   1:  PR[91] = PR[90];
   1:  PR[91,1] = PR[90,1] + 58.395;
   1:  PR[91,2] = PR[90,2] + 13.062;
   1:  PR[91,3] = PR[90,3] + 26.195;
   1:  PR[92] = PR[91];
   1:  PR[92,3] = PR[92,3] + 20;
   1:J PR[92] 10% FINE;
   1:L PR[91] R[100]mm/sec CNT100;
   1:  CALL LASER_DRAHT_START;
   1:  PR[91,1] = PR[90,1] + 56.578;
   1:  PR[91,2] = PR[90,2] + 11.493;
   1:L PR[91] R[100]mm/sec CNT100;
   1:  PR[91,1] = PR[90,1] + 55.757;
   1:  PR[91,2] = PR[90,2] + 10.310;
   1:L PR[91] R[100]mm/sec CNT100;
   1:  PR[91,1] = PR[90,1] + 53.974;
   1:  PR[91,2] = PR[90,2] + 7.827;
   1:L PR[91] R[100]mm/sec CNT100;
   1:  PR[91,1] = PR[90,1] + 52.340;
   1:  PR[91,2] = PR[90,2] + 3.681;
   1:L PR[91] R[100]mm/sec CNT100;
   1:  PR[91,1] = PR[90,1] + 52.290;
   1:  PR[91,2] = PR[90,2] + 3.287;
   1:L PR[91] R[100]mm/sec CNT100;
   1:  PR[91,1] = PR[90,1] + 52.250;
   1:  PR[91,2] = PR[90,2] + 2.641;
   1:L PR[91] R[100]mm/sec CNT100;
   1:  PR[91,1] = PR[90,1] + 51.813;
   1:  PR[91,2] = PR[90,2] + -0.787;
   1:L PR[91] R[100]mm/sec CNT100;
   1:  PR[91,1] = PR[90,1] + 51.829;
   1:  PR[91,2] = PR[90,2] + -1.013;
   1:L PR[91] R[100]mm/sec CNT100;
   1:  PR[91,1] = PR[90,1] + 52.341;
   1:  PR[91,2] = PR[90,2] + -5.143;
   1:L PR[91] R[100]mm/sec CNT100;
   1:  PR[91,1] = PR[90,1] + 53.979;
   1:  PR[91,2] = PR[90,2] + -9.300;
   1:L PR[91] R[100]mm/sec CNT100;
   1:  PR[91,1] = PR[90,1] + 54.599;
   1:  PR[91,2] = PR[90,2] + -10.189;
   1:L PR[91] R[100]mm/sec CNT100;
   1:  PR[91,1] = PR[90,1] + 56.578;
   1:  PR[91,2] = PR[90,2] + -12.957;
   1:L PR[91] R[100]mm/sec CNT100;
   1:  PR[91,1] = PR[90,1] + 57.989;
   1:  PR[91,2] = PR[90,2] + -14.220;
   1:L PR[91] R[100]mm/sec CNT100;
   1:  PR[91,1] = PR[90,1] + 59.963;
   1:  PR[91,2] = PR[90,2] + -15.936;
   1:L PR[91] R[100]mm/sec CNT100;
   1:  PR[91,1] = PR[90,1] + 62.463;
   1:  PR[91,2] = PR[90,2] + -17.317;
   1:L PR[91] R[100]mm/sec CNT100;
   1:  PR[91,1] = PR[90,1] + 63.933;
   1:  PR[91,2] = PR[90,2] + -18.100;
   1:L PR[91] R[100]mm/sec CNT100;
   1:  PR[91,1] = PR[90,1] + 67.611;
   1:  PR[91,2] = PR[90,2] + -19.179;
   1:L PR[91] R[100]mm/sec CNT100;
   1:  PR[91,1] = PR[90,1] + 68.271;
   1:  PR[91,2] = PR[90,2] + -19.362;
   1:L PR[91] R[100]mm/sec CNT100;
   1:  PR[91,1] = PR[90,1] + 72.776;
   1:  PR[91,2] = PR[90,2] + -19.685;
   1:L PR[91] R[100]mm/sec CNT100;
   1:  PR[91,1] = PR[90,1] + 77.061;
   1:  PR[91,2] = PR[90,2] + -19.105;
   1:L PR[91] R[100]mm/sec CNT100;
   1:  PR[91,1] = PR[90,1] + 81.078;
   1:  PR[91,2] = PR[90,2] + -17.631;
   1:L PR[91] R[100]mm/sec CNT100;
   1:  PR[91,1] = PR[90,1] + 84.652;
   1:  PR[91,2] = PR[90,2] + -15.336;
   1:L PR[91] R[100]mm/sec CNT100;
   1:  PR[91,1] = PR[90,1] + 87.617;
   1:  PR[91,2] = PR[90,2] + -12.341;
   1:L PR[91] R[100]mm/sec CNT100;
   1:  PR[91,1] = PR[90,1] + 89.839;
   1:  PR[91,2] = PR[90,2] + -8.790;
   1:L PR[91] R[100]mm/sec CNT100;
   1:  PR[91,1] = PR[90,1] + 90.385;
   1:  PR[91,2] = PR[90,2] + -7.237;
   1:L PR[91] R[100]mm/sec CNT100;
   1:  PR[91,1] = PR[90,1] + 91.211;
   1:  PR[91,2] = PR[90,2] + -4.857;
   1:L PR[91] R[100]mm/sec CNT100;
   1:  PR[91,1] = PR[90,1] + 91.419;
   1:  PR[91,2] = PR[90,2] + -3.053;
   1:L PR[91] R[100]mm/sec CNT100;
   1:  PR[91,1] = PR[90,1] + 91.779;
   1:  PR[91,2] = PR[90,2] + -0.692;
   1:L PR[91] R[100]mm/sec CNT100;
   1:  PR[91,1] = PR[90,1] + 91.764;
   1:  PR[91,2] = PR[90,2] + -0.562;
   1:L PR[91] R[100]mm/sec CNT100;
   1:  PR[91,1] = PR[90,1] + 91.478;
   1:  PR[91,2] = PR[90,2] + 0.980;
   1:L PR[91] R[100]mm/sec CNT100;
   1:  PR[91,1] = PR[90,1] + 91.210;
   1:  PR[91,2] = PR[90,2] + 3.401;
   1:L PR[91] R[100]mm/sec CNT100;
   1:  PR[91,1] = PR[90,1] + 89.838;
   1:  PR[91,2] = PR[90,2] + 7.333;
   1:L PR[91] R[100]mm/sec CNT100;
   1:  PR[91,1] = PR[90,1] + 87.617;
   1:  PR[91,2] = PR[90,2] + 10.882;
   1:L PR[91] R[100]mm/sec CNT100;
   1:  PR[91,1] = PR[90,1] + 84.658;
   1:  PR[91,2] = PR[90,2] + 13.872;
   1:L PR[91] R[100]mm/sec CNT100;
   1:  PR[91,1] = PR[90,1] + 83.729;
   1:  PR[91,2] = PR[90,2] + 14.458;
   1:L PR[91] R[100]mm/sec CNT100;
   1:  PR[91,1] = PR[90,1] + 81.076;
   1:  PR[91,2] = PR[90,2] + 16.173;
   1:L PR[91] R[100]mm/sec CNT100;
   1:  PR[91,1] = PR[90,1] + 77.061;
   1:  PR[91,2] = PR[90,2] + 17.647;
   1:L PR[91] R[100]mm/sec CNT100;
   1:  PR[91,1] = PR[90,1] + 72.779;
   1:  PR[91,2] = PR[90,2] + 18.226;
   1:L PR[91] R[100]mm/sec CNT100;
   1:  PR[91,1] = PR[90,1] + 68.646;
   1:  PR[91,2] = PR[90,2] + 17.919;
   1:L PR[91] R[100]mm/sec CNT100;
   1:  PR[91,1] = PR[90,1] + 68.271;
   1:  PR[91,2] = PR[90,2] + 17.899;
   1:L PR[91] R[100]mm/sec CNT100;
   1:  PR[91,1] = PR[90,1] + 64.923;
   1:  PR[91,2] = PR[90,2] + 16.906;
   1:L PR[91] R[100]mm/sec CNT100;
   1:  PR[91,1] = PR[90,1] + 63.934;
   1:  PR[91,2] = PR[90,2] + 16.636;
   1:L PR[91] R[100]mm/sec CNT100;
   1:  PR[91,1] = PR[90,1] + 61.478;
   1:  PR[91,2] = PR[90,2] + 15.271;
   1:L PR[91] R[100]mm/sec CNT100;
   1:  PR[91,1] = PR[90,1] + 59.964;
   1:  PR[91,2] = PR[90,2] + 14.472;
   1:L PR[91] R[100]mm/sec CNT100;
   1:  PR[91,1] = PR[90,1] + 58.395;
   1:  PR[91,2] = PR[90,2] + 13.062;
   1:L PR[91] R[100]mm/sec CNT100TB   .50sec,CALL END_PUD;
   1:  PR[92] = PR[91];
   1:  PR[92,3] = PR[92,3] + 20;
   1:J PR[92] 10% FINE;
   1:  PR[91,1] = PR[90,1] + 41.160;
   1:  PR[91,2] = PR[90,2] + 8.184;
   1:  PR[92] = PR[91];
   1:  PR[92,3] = PR[92,3] + 20;
   1:J PR[92] 10% FINE;
   1:L PR[91] R[100]mm/sec CNT100;
   1:  CALL LASER_DRAHT_START;
   1:  PR[91,1] = PR[90,1] + 40.947;
   1:  PR[91,2] = PR[90,2] + 8.666;
   1:L PR[91] R[100]mm/sec CNT100;
   1:  PR[91,1] = PR[90,1] + 38.341;
   1:  PR[91,2] = PR[90,2] + 12.079;
   1:L PR[91] R[100]mm/sec CNT100;
   1:  PR[91,1] = PR[90,1] + 37.898;
   1:  PR[91,2] = PR[90,2] + 12.643;
   1:L PR[91] R[100]mm/sec CNT100;
   1:  PR[91,1] = PR[90,1] + 33.979;
   1:  PR[91,2] = PR[90,2] + 15.652;
   1:L PR[91] R[100]mm/sec CNT100;
   1:  PR[91,1] = PR[90,1] + 30.208;
   1:  PR[91,2] = PR[90,2] + 17.229;
   1:L PR[91] R[100]mm/sec CNT100;
   1:  PR[91,1] = PR[90,1] + 29.432;
   1:  PR[91,2] = PR[90,2] + 17.545;
   1:L PR[91] R[100]mm/sec CNT100;
   1:  PR[91,1] = PR[90,1] + 24.528;
   1:  PR[91,2] = PR[90,2] + 18.204;
   1:L PR[91] R[100]mm/sec CNT100;
   1:  PR[91,1] = PR[90,1] + 19.621;
   1:  PR[91,2] = PR[90,2] + 17.571;
   1:L PR[91] R[100]mm/sec CNT100;
   1:  PR[91,1] = PR[90,1] + 16.027;
   1:  PR[91,2] = PR[90,2] + 16.100;
   1:L PR[91] R[100]mm/sec CNT100;
   1:  PR[91,1] = PR[90,1] + 15.045;
   1:  PR[91,2] = PR[90,2] + 15.693;
   1:L PR[91] R[100]mm/sec CNT100;
   1:  PR[91,1] = PR[90,1] + 11.102;
   1:  PR[91,2] = PR[90,2] + 12.688;
   1:L PR[91] R[100]mm/sec CNT100;
   1:  PR[91,1] = PR[90,1] + 8.076;
   1:  PR[91,2] = PR[90,2] + 8.763;
   1:L PR[91] R[100]mm/sec CNT100;
   1:  PR[91,1] = PR[90,1] + 6.171;
   1:  PR[91,2] = PR[90,2] + 4.186;
   1:L PR[91] R[100]mm/sec CNT100;
   1:  PR[91,1] = PR[90,1] + 5.520;
   1:  PR[91,2] = PR[90,2] + -0.729;
   1:L PR[91] R[100]mm/sec CNT100;
   1:  PR[91,1] = PR[90,1] + 6.171;
   1:  PR[91,2] = PR[90,2] + -5.646;
   1:L PR[91] R[100]mm/sec CNT100;
   1:  PR[91,1] = PR[90,1] + 8.077;
   1:  PR[91,2] = PR[90,2] + -10.225;
   1:L PR[91] R[100]mm/sec CNT100;
   1:  PR[91,1] = PR[90,1] + 11.105;
   1:  PR[91,2] = PR[90,2] + -14.150;
   1:L PR[91] R[100]mm/sec CNT100;
   1:  PR[91,1] = PR[90,1] + 15.047;
   1:  PR[91,2] = PR[90,2] + -17.153;
   1:L PR[91] R[100]mm/sec CNT100;
   1:  PR[91,1] = PR[90,1] + 19.631;
   1:  PR[91,2] = PR[90,2] + -19.033;
   1:L PR[91] R[100]mm/sec CNT100;
   1:  PR[91,1] = PR[90,1] + 20.613;
   1:  PR[91,2] = PR[90,2] + -19.162;
   1:L PR[91] R[100]mm/sec CNT100;
   1:  PR[91,1] = PR[90,1] + 24.534;
   1:  PR[91,2] = PR[90,2] + -19.663;
   1:L PR[91] R[100]mm/sec CNT100;
   1:  PR[91,1] = PR[90,1] + 29.431;
   1:  PR[91,2] = PR[90,2] + -19.003;
   1:L PR[91] R[100]mm/sec CNT100;
   1:  PR[91,1] = PR[90,1] + 33.994;
   1:  PR[91,2] = PR[90,2] + -17.103;
   1:L PR[91] R[100]mm/sec CNT100;
   1:  PR[91,1] = PR[90,1] + 34.610;
   1:  PR[91,2] = PR[90,2] + -16.637;
   1:L PR[91] R[100]mm/sec CNT100;
   1:  PR[91,1] = PR[90,1] + 37.894;
   1:  PR[91,2] = PR[90,2] + -14.104;
   1:L PR[91] R[100]mm/sec CNT100;
   1:  PR[91,1] = PR[90,1] + 40.936;
   1:  PR[91,2] = PR[90,2] + -10.139;
   1:L PR[91] R[100]mm/sec CNT100;
   1:  PR[91,1] = PR[90,1] + 42.580;
   1:  PR[91,2] = PR[90,2] + -6.157;
   1:L PR[91] R[100]mm/sec CNT100;
   1:  PR[91,1] = PR[90,1] + 42.727;
   1:  PR[91,2] = PR[90,2] + -5.828;
   1:L PR[91] R[100]mm/sec CNT100;
   1:  PR[91,1] = PR[90,1] + 42.869;
   1:  PR[91,2] = PR[90,2] + -5.270;
   1:L PR[91] R[100]mm/sec CNT100;
   1:  PR[91,1] = PR[90,1] + 43.360;
   1:  PR[91,2] = PR[90,2] + -1.542;
   1:L PR[91] R[100]mm/sec CNT100;
   1:  PR[91,1] = PR[90,1] + 43.428;
   1:  PR[91,2] = PR[90,2] + -0.772;
   1:L PR[91] R[100]mm/sec CNT100;
   1:  PR[91,1] = PR[90,1] + 42.958;
   1:  PR[91,2] = PR[90,2] + 2.798;
   1:L PR[91] R[100]mm/sec CNT100;
   1:  PR[91,1] = PR[90,1] + 42.866;
   1:  PR[91,2] = PR[90,2] + 3.815;
   1:L PR[91] R[100]mm/sec CNT100;
   1:  PR[91,1] = PR[90,1] + 42.702;
   1:  PR[91,2] = PR[90,2] + 4.446;
   1:L PR[91] R[100]mm/sec CNT100;
   1:  PR[91,1] = PR[90,1] + 41.160;
   1:  PR[91,2] = PR[90,2] + 8.184;
   1:L PR[91] R[100]mm/sec CNT100TB   .50sec,CALL END_PUD;
   1:  PR[92] = PR[91];
   1:  PR[92,3] = PR[92,3] + 20;
   1:J PR[92] 10% FINE;
   1:  PR[91,1] = PR[90,1] + -27.836;
   1:  PR[91,2] = PR[90,2] + -18.849;
   1:  PR[92] = PR[91];
   1:  PR[92,3] = PR[92,3] + 20;
   1:J PR[92] 10% FINE;
   1:L PR[91] R[100]mm/sec CNT100;
   1:  CALL LASER_DRAHT_START;
   1:  PR[91,1] = PR[90,1] + -25.440;
   1:  PR[91,2] = PR[90,2] + -19.136;
   1:L PR[91] R[100]mm/sec CNT100;
   1:  PR[91,1] = PR[90,1] + -23.651;
   1:  PR[91,2] = PR[90,2] + -19.368;
   1:L PR[91] R[100]mm/sec CNT100;
   1:  PR[91,1] = PR[90,1] + -21.486;
   1:  PR[91,2] = PR[90,2] + -19.143;
   1:L PR[91] R[100]mm/sec CNT100;
   1:  PR[91,1] = PR[90,1] + -19.442;
   1:  PR[91,2] = PR[90,2] + -18.953;
   1:L PR[91] R[100]mm/sec CNT100;
   1:  PR[91,1] = PR[90,1] + -17.618;
   1:  PR[91,2] = PR[90,2] + -18.338;
   1:L PR[91] R[100]mm/sec CNT100;
   1:  PR[91,1] = PR[90,1] + -15.419;
   1:  PR[91,2] = PR[90,2] + -17.622;
   1:L PR[91] R[100]mm/sec CNT100;
   1:  PR[91,1] = PR[90,1] + -13.998;
   1:  PR[91,2] = PR[90,2] + -16.752;
   1:L PR[91] R[100]mm/sec CNT100;
   1:  PR[91,1] = PR[90,1] + -11.783;
   1:  PR[91,2] = PR[90,2] + -15.426;
   1:L PR[91] R[100]mm/sec CNT100;
   1:  PR[91,1] = PR[90,1] + -8.736;
   1:  PR[91,2] = PR[90,2] + -12.480;
   1:L PR[91] R[100]mm/sec CNT100;
   1:  PR[91,1] = PR[90,1] + -6.429;
   1:  PR[91,2] = PR[90,2] + -8.922;
   1:L PR[91] R[100]mm/sec CNT100;
   1:  PR[91,1] = PR[90,1] + -4.997;
   1:  PR[91,2] = PR[90,2] + -4.946;
   1:L PR[91] R[100]mm/sec CNT100;
   1:  PR[91,1] = PR[90,1] + -4.548;
   1:  PR[91,2] = PR[90,2] + -0.738;
   1:L PR[91] R[100]mm/sec CNT100;
   1:  PR[91,1] = PR[90,1] + -4.635;
   1:  PR[91,2] = PR[90,2] + 0.012;
   1:L PR[91] R[100]mm/sec CNT100;
   1:  PR[91,1] = PR[90,1] + -4.624;
   1:  PR[91,2] = PR[90,2] + 0.292;
   1:L PR[91] R[100]mm/sec CNT100;
   1:  PR[91,1] = PR[90,1] + -4.994;
   1:  PR[91,2] = PR[90,2] + 3.478;
   1:L PR[91] R[100]mm/sec CNT100;
   1:  PR[91,1] = PR[90,1] + -6.429;
   1:  PR[91,2] = PR[90,2] + 7.463;
   1:L PR[91] R[100]mm/sec CNT100;
   1:  PR[91,1] = PR[90,1] + -8.736;
   1:  PR[91,2] = PR[90,2] + 11.021;
   1:L PR[91] R[100]mm/sec CNT100;
   1:  PR[91,1] = PR[90,1] + -11.790;
   1:  PR[91,2] = PR[90,2] + 13.974;
   1:L PR[91] R[100]mm/sec CNT100;
   1:  PR[91,1] = PR[90,1] + -13.095;
   1:  PR[91,2] = PR[90,2] + 14.772;
   1:L PR[91] R[100]mm/sec CNT100;
   1:  PR[91,1] = PR[90,1] + -15.419;
   1:  PR[91,2] = PR[90,2] + 16.165;
   1:L PR[91] R[100]mm/sec CNT100;
   1:  PR[91,1] = PR[90,1] + -17.136;
   1:  PR[91,2] = PR[90,2] + 16.744;
   1:L PR[91] R[100]mm/sec CNT100;
   1:  PR[91,1] = PR[90,1] + -19.442;
   1:  PR[91,2] = PR[90,2] + 17.497;
   1:L PR[91] R[100]mm/sec CNT100;
   1:  PR[91,1] = PR[90,1] + -21.527;
   1:  PR[91,2] = PR[90,2] + 17.713;
   1:L PR[91] R[100]mm/sec CNT100;
   1:  PR[91,1] = PR[90,1] + -23.651;
   1:  PR[91,2] = PR[90,2] + 17.912;
   1:L PR[91] R[100]mm/sec CNT100;
   1:  PR[91,1] = PR[90,1] + -25.996;
   1:  PR[91,2] = PR[90,2] + 17.631;
   1:L PR[91] R[100]mm/sec CNT100;
   1:  PR[91,1] = PR[90,1] + -27.833;
   1:  PR[91,2] = PR[90,2] + 17.393;
   1:L PR[91] R[100]mm/sec CNT100;
   1:  PR[91,1] = PR[90,1] + -31.795;
   1:  PR[91,2] = PR[90,2] + 15.974;
   1:L PR[91] R[100]mm/sec CNT100;
   1:  PR[91,1] = PR[90,1] + -34.157;
   1:  PR[91,2] = PR[90,2] + 14.483;
   1:L PR[91] R[100]mm/sec CNT100;
   1:  PR[91,1] = PR[90,1] + -35.320;
   1:  PR[91,2] = PR[90,2] + 13.736;
   1:L PR[91] R[100]mm/sec CNT100;
   1:  PR[91,1] = PR[90,1] + -38.261;
   1:  PR[91,2] = PR[90,2] + 10.783;
   1:L PR[91] R[100]mm/sec CNT100;
   1:  PR[91,1] = PR[90,1] + -40.465;
   1:  PR[91,2] = PR[90,2] + 7.271;
   1:L PR[91] R[100]mm/sec CNT100;
   1:  PR[91,1] = PR[90,1] + -41.829;
   1:  PR[91,2] = PR[90,2] + 3.370;
   1:L PR[91] R[100]mm/sec CNT100;
   1:  PR[91,1] = PR[90,1] + -42.198;
   1:  PR[91,2] = PR[90,2] + 0.121;
   1:L PR[91] R[100]mm/sec CNT100;
   1:  PR[91,1] = PR[90,1] + -42.279;
   1:  PR[91,2] = PR[90,2] + -0.278;
   1:L PR[91] R[100]mm/sec CNT100;
   1:  PR[91,1] = PR[90,1] + -42.329;
   1:  PR[91,2] = PR[90,2] + -0.717;
   1:L PR[91] R[100]mm/sec CNT100;
   1:  PR[91,1] = PR[90,1] + -41.936;
   1:  PR[91,2] = PR[90,2] + -3.871;
   1:L PR[91] R[100]mm/sec CNT100;
   1:  PR[91,1] = PR[90,1] + -41.829;
   1:  PR[91,2] = PR[90,2] + -4.830;
   1:L PR[91] R[100]mm/sec CNT100;
   1:  PR[91,1] = PR[90,1] + -40.465;
   1:  PR[91,2] = PR[90,2] + -8.730;
   1:L PR[91] R[100]mm/sec CNT100;
   1:  PR[91,1] = PR[90,1] + -38.261;
   1:  PR[91,2] = PR[90,2] + -12.242;
   1:L PR[91] R[100]mm/sec CNT100;
   1:  PR[91,1] = PR[90,1] + -35.324;
   1:  PR[91,2] = PR[90,2] + -15.192;
   1:L PR[91] R[100]mm/sec CNT100;
   1:  PR[91,1] = PR[90,1] + -31.796;
   1:  PR[91,2] = PR[90,2] + -17.431;
   1:L PR[91] R[100]mm/sec CNT100;
   1:  PR[91,1] = PR[90,1] + -29.320;
   1:  PR[91,2] = PR[90,2] + -18.308;
   1:L PR[91] R[100]mm/sec CNT100;
   1:  PR[91,1] = PR[90,1] + -27.836;
   1:  PR[91,2] = PR[90,2] + -18.849;
   1:L PR[91] R[100]mm/sec CNT100TB   .50sec,CALL END_PUD;
   1:  PR[92] = PR[91];
   1:  PR[92,3] = PR[92,3] + 20;
   1:J PR[92] 10% FINE;
   1:  PR[91,1] = PR[90,1] + -59.903;
   1:  PR[91,2] = PR[90,2] + 13.243;
   1:  PR[92] = PR[91];
   1:  PR[92,3] = PR[92,3] + 20;
   1:J PR[92] 10% FINE;
   1:L PR[91] R[100]mm/sec CNT100;
   1:  CALL LASER_DRAHT_START;
   1:  PR[91,1] = PR[90,1] + -63.277;
   1:  PR[91,2] = PR[90,2] + 15.489;
   1:L PR[91] R[100]mm/sec CNT100;
   1:  PR[91,1] = PR[90,1] + -67.051;
   1:  PR[91,2] = PR[90,2] + 17.006;
   1:L PR[91] R[100]mm/sec CNT100;
   1:  PR[91,1] = PR[90,1] + -71.057;
   1:  PR[91,2] = PR[90,2] + 17.738;
   1:L PR[91] R[100]mm/sec CNT100;
   1:  PR[91,1] = PR[90,1] + -75.056;
   1:  PR[91,2] = PR[90,2] + 17.673;
   1:L PR[91] R[100]mm/sec CNT100;
   1:  PR[91,1] = PR[90,1] + -78.887;
   1:  PR[91,2] = PR[90,2] + 16.820;
   1:L PR[91] R[100]mm/sec CNT100;
   1:  PR[91,1] = PR[90,1] + -82.443;
   1:  PR[91,2] = PR[90,2] + 15.213;
   1:L PR[91] R[100]mm/sec CNT100;
   1:  PR[91,1] = PR[90,1] + -85.580;
   1:  PR[91,2] = PR[90,2] + 12.923;
   1:L PR[91] R[100]mm/sec CNT100;
   1:  PR[91,1] = PR[90,1] + -88.164;
   1:  PR[91,2] = PR[90,2] + 10.051;
   1:L PR[91] R[100]mm/sec CNT100;
   1:  PR[91,1] = PR[90,1] + -90.091;
   1:  PR[91,2] = PR[90,2] + 6.722;
   1:L PR[91] R[100]mm/sec CNT100;
   1:  PR[91,1] = PR[90,1] + -91.279;
   1:  PR[91,2] = PR[90,2] + 3.075;
   1:L PR[91] R[100]mm/sec CNT100;
   1:  PR[91,1] = PR[90,1] + -91.449;
   1:  PR[91,2] = PR[90,2] + 1.478;
   1:L PR[91] R[100]mm/sec CNT100;
   1:  PR[91,1] = PR[90,1] + -91.504;
   1:  PR[91,2] = PR[90,2] + 1.218;
   1:L PR[91] R[100]mm/sec CNT100;
   1:  PR[91,1] = PR[90,1] + -91.792;
   1:  PR[91,2] = PR[90,2] + -0.720;
   1:L PR[91] R[100]mm/sec CNT100;
   1:  PR[91,1] = PR[90,1] + -91.545;
   1:  PR[91,2] = PR[90,2] + -2.284;
   1:L PR[91] R[100]mm/sec CNT100;
   1:  PR[91,1] = PR[90,1] + -91.428;
   1:  PR[91,2] = PR[90,2] + -2.781;
   1:L PR[91] R[100]mm/sec CNT100;
   1:  PR[91,1] = PR[90,1] + -91.245;
   1:  PR[91,2] = PR[90,2] + -4.536;
   1:L PR[91] R[100]mm/sec CNT100;
   1:  PR[91,1] = PR[90,1] + -90.580;
   1:  PR[91,2] = PR[90,2] + -6.563;
   1:L PR[91] R[100]mm/sec CNT100;
   1:  PR[91,1] = PR[90,1] + -90.054;
   1:  PR[91,2] = PR[90,2] + -8.183;
   1:L PR[91] R[100]mm/sec CNT100;
   1:  PR[91,1] = PR[90,1] + -88.122;
   1:  PR[91,2] = PR[90,2] + -11.513;
   1:L PR[91] R[100]mm/sec CNT100;
   1:  PR[91,1] = PR[90,1] + -85.530;
   1:  PR[91,2] = PR[90,2] + -14.388;
   1:L PR[91] R[100]mm/sec CNT100;
   1:  PR[91,1] = PR[90,1] + -82.382;
   1:  PR[91,2] = PR[90,2] + -16.682;
   1:L PR[91] R[100]mm/sec CNT100;
   1:  PR[91,1] = PR[90,1] + -78.812;
   1:  PR[91,2] = PR[90,2] + -18.295;
   1:L PR[91] R[100]mm/sec CNT100;
   1:  PR[91,1] = PR[90,1] + -74.967;
   1:  PR[91,2] = PR[90,2] + -19.151;
   1:L PR[91] R[100]mm/sec CNT100;
   1:  PR[91,1] = PR[90,1] + -71.014;
   1:  PR[91,2] = PR[90,2] + -19.210;
   1:L PR[91] R[100]mm/sec CNT100;
   1:  PR[91,1] = PR[90,1] + -67.120;
   1:  PR[91,2] = PR[90,2] + -18.462;
   1:L PR[91] R[100]mm/sec CNT100;
   1:  PR[91,1] = PR[90,1] + -65.650;
   1:  PR[91,2] = PR[90,2] + -17.846;
   1:L PR[91] R[100]mm/sec CNT100;
   1:  PR[91,1] = PR[90,1] + -63.333;
   1:  PR[91,2] = PR[90,2] + -16.929;
   1:L PR[91] R[100]mm/sec CNT100;
   1:  PR[91,1] = PR[90,1] + -59.926;
   1:  PR[91,2] = PR[90,2] + -14.691;
   1:L PR[91] R[100]mm/sec CNT100;
   1:  PR[91,1] = PR[90,1] + -57.766;
   1:  PR[91,2] = PR[90,2] + -12.491;
   1:L PR[91] R[100]mm/sec CNT100;
   1:  PR[91,1] = PR[90,1] + -57.074;
   1:  PR[91,2] = PR[90,2] + -11.805;
   1:L PR[91] R[100]mm/sec CNT100;
   1:  PR[91,1] = PR[90,1] + -55.664;
   1:  PR[91,2] = PR[90,2] + -9.558;
   1:L PR[91] R[100]mm/sec CNT100;
   1:  PR[91,1] = PR[90,1] + -54.929;
   1:  PR[91,2] = PR[90,2] + -8.413;
   1:L PR[91] R[100]mm/sec CNT100;
   1:  PR[91,1] = PR[90,1] + -53.599;
   1:  PR[91,2] = PR[90,2] + -4.666;
   1:L PR[91] R[100]mm/sec CNT100;
   1:  PR[91,1] = PR[90,1] + -53.360;
   1:  PR[91,2] = PR[90,2] + -2.607;
   1:L PR[91] R[100]mm/sec CNT100;
   1:  PR[91,1] = PR[90,1] + -53.225;
   1:  PR[91,2] = PR[90,2] + -0.745;
   1:L PR[91] R[100]mm/sec CNT100;
   1:  PR[91,1] = PR[90,1] + -53.308;
   1:  PR[91,2] = PR[90,2] + 0.189;
   1:L PR[91] R[100]mm/sec CNT100;
   1:  PR[91,1] = PR[90,1] + -53.649;
   1:  PR[91,2] = PR[90,2] + 3.212;
   1:L PR[91] R[100]mm/sec CNT100;
   1:  PR[91,1] = PR[90,1] + -54.966;
   1:  PR[91,2] = PR[90,2] + 6.966;
   1:L PR[91] R[100]mm/sec CNT100;
   1:  PR[91,1] = PR[90,1] + -57.088;
   1:  PR[91,2] = PR[90,2] + 10.361;
   1:L PR[91] R[100]mm/sec CNT100;
   1:  PR[91,1] = PR[90,1] + -59.903;
   1:  PR[91,2] = PR[90,2] + 13.243;
   1:L PR[91] R[100]mm/sec CNT100TB   .50sec,CALL END_PUD;
   1:  PR[92] = PR[91];
   1:  PR[92,3] = PR[92,3] + 20;
   1:J PR[92] 10% FINE;
   1:  PR[91] = PR[90];
   1:  PR[91,1] = PR[90,1] + 91.045;
   1:  PR[91,2] = PR[90,2] + 3.417;
   1:  PR[91,3] = PR[90,3] + 27.495;
   1:  PR[92] = PR[91];
   1:  PR[92,3] = PR[92,3] + 20;
   1:J PR[92] 10% FINE;
   1:L PR[91] R[100]mm/sec CNT100;
   1:  CALL LASER_DRAHT_START;
   1:  PR[91,1] = PR[90,1] + 89.670;
   1:  PR[91,2] = PR[90,2] + 7.365;
   1:L PR[91] R[100]mm/sec CNT100;
   1:  PR[91,1] = PR[90,1] + 87.443;
   1:  PR[91,2] = PR[90,2] + 10.931;
   1:L PR[91] R[100]mm/sec CNT100;
   1:  PR[91,1] = PR[90,1] + 84.468;
   1:  PR[91,2] = PR[90,2] + 13.943;
   1:L PR[91] R[100]mm/sec CNT100;
   1:  PR[91,1] = PR[90,1] + 80.881;
   1:  PR[91,2] = PR[90,2] + 16.252;
   1:L PR[91] R[100]mm/sec CNT100;
   1:  PR[91,1] = PR[90,1] + 76.821;
   1:  PR[91,2] = PR[90,2] + 17.748;
   1:L PR[91] R[100]mm/sec CNT100;
   1:  PR[91,1] = PR[90,1] + 72.793;
   1:  PR[91,2] = PR[90,2] + 18.312;
   1:L PR[91] R[100]mm/sec CNT100;
   1:  PR[91,1] = PR[90,1] + 72.358;
   1:  PR[91,2] = PR[90,2] + 18.382;
   1:L PR[91] R[100]mm/sec CNT100;
   1:  PR[91,1] = PR[90,1] + 68.913;
   1:  PR[91,2] = PR[90,2] + 18.126;
   1:L PR[91] R[100]mm/sec CNT100;
   1:  PR[91,1] = PR[90,1] + 67.834;
   1:  PR[91,2] = PR[90,2] + 18.069;
   1:L PR[91] R[100]mm/sec CNT100;
   1:  PR[91,1] = PR[90,1] + 65.170;
   1:  PR[91,2] = PR[90,2] + 17.279;
   1:L PR[91] R[100]mm/sec CNT100;
   1:  PR[91,1] = PR[90,1] + 63.449;
   1:  PR[91,2] = PR[90,2] + 16.811;
   1:L PR[91] R[100]mm/sec CNT100;
   1:  PR[91,1] = PR[90,1] + 61.667;
   1:  PR[91,2] = PR[90,2] + 15.820;
   1:L PR[91] R[100]mm/sec CNT100;
   1:  PR[91,1] = PR[90,1] + 59.428;
   1:  PR[91,2] = PR[90,2] + 14.638;
   1:L PR[91] R[100]mm/sec CNT100;
   1:  PR[91,1] = PR[90,1] + 58.480;
   1:  PR[91,2] = PR[90,2] + 13.786;
   1:L PR[91] R[100]mm/sec CNT100;
   1:  PR[91,1] = PR[90,1] + 55.992;
   1:  PR[91,2] = PR[90,2] + 11.637;
   1:L PR[91] R[100]mm/sec CNT100;
   1:  PR[91,1] = PR[90,1] + 55.687;
   1:  PR[91,2] = PR[90,2] + 11.198;
   1:L PR[91] R[100]mm/sec CNT100;
   1:  PR[91,1] = PR[90,1] + 53.343;
   1:  PR[91,2] = PR[90,2] + 7.934;
   1:L PR[91] R[100]mm/sec CNT100;
   1:  PR[91,1] = PR[90,1] + 52.852;
   1:  PR[91,2] = PR[90,2] + 6.692;
   1:L PR[91] R[100]mm/sec CNT100;
   1:  PR[91,1] = PR[90,1] + 51.596;
   1:  PR[91,2] = PR[90,2] + 3.729;
   1:L PR[91] R[100]mm/sec CNT100;
   1:  PR[91,1] = PR[90,1] + 51.566;
   1:  PR[91,2] = PR[90,2] + 3.532;
   1:L PR[91] R[100]mm/sec CNT100;
   1:  PR[91,1] = PR[90,1] + 50.974;
   1:  PR[91,2] = PR[90,2] + -0.729;
   1:L PR[91] R[100]mm/sec CNT100;
   1:  PR[91,1] = PR[90,1] + 51.566;
   1:  PR[91,2] = PR[90,2] + -4.991;
   1:L PR[91] R[100]mm/sec CNT100;
   1:  PR[91,1] = PR[90,1] + 51.596;
   1:  PR[91,2] = PR[90,2] + -5.188;
   1:L PR[91] R[100]mm/sec CNT100;
   1:  PR[91,1] = PR[90,1] + 52.852;
   1:  PR[91,2] = PR[90,2] + -8.151;
   1:L PR[91] R[100]mm/sec CNT100;
   1:  PR[91,1] = PR[90,1] + 53.344;
   1:  PR[91,2] = PR[90,2] + -9.395;
   1:L PR[91] R[100]mm/sec CNT100;
   1:  PR[91,1] = PR[90,1] + 55.992;
   1:  PR[91,2] = PR[90,2] + -13.102;
   1:L PR[91] R[100]mm/sec CNT100;
   1:  PR[91,1] = PR[90,1] + 56.547;
   1:  PR[91,2] = PR[90,2] + -13.598;
   1:L PR[91] R[100]mm/sec CNT100;
   1:  PR[91,1] = PR[90,1] + 59.428;
   1:  PR[91,2] = PR[90,2] + -16.102;
   1:L PR[91] R[100]mm/sec CNT100;
   1:  PR[91,1] = PR[90,1] + 60.964;
   1:  PR[91,2] = PR[90,2] + -16.951;
   1:L PR[91] R[100]mm/sec CNT100;
   1:  PR[91,1] = PR[90,1] + 63.449;
   1:  PR[91,2] = PR[90,2] + -18.274;
   1:L PR[91] R[100]mm/sec CNT100;
   1:  PR[91,1] = PR[90,1] + 66.138;
   1:  PR[91,2] = PR[90,2] + -19.063;
   1:L PR[91] R[100]mm/sec CNT100;
   1:  PR[91,1] = PR[90,1] + 67.834;
   1:  PR[91,2] = PR[90,2] + -19.532;
   1:L PR[91] R[100]mm/sec CNT100;
   1:  PR[91,1] = PR[90,1] + 71.592;
   1:  PR[91,2] = PR[90,2] + -19.801;
   1:L PR[91] R[100]mm/sec CNT100;
   1:  PR[91,1] = PR[90,1] + 72.358;
   1:  PR[91,2] = PR[90,2] + -19.844;
   1:L PR[91] R[100]mm/sec CNT100;
   1:  PR[91,1] = PR[90,1] + 76.818;
   1:  PR[91,2] = PR[90,2] + -19.208;
   1:L PR[91] R[100]mm/sec CNT100;
   1:  PR[91,1] = PR[90,1] + 80.881;
   1:  PR[91,2] = PR[90,2] + -17.711;
   1:L PR[91] R[100]mm/sec CNT100;
   1:  PR[91,1] = PR[90,1] + 84.468;
   1:  PR[91,2] = PR[90,2] + -15.401;
   1:L PR[91] R[100]mm/sec CNT100;
   1:  PR[91,1] = PR[90,1] + 87.446;
   1:  PR[91,2] = PR[90,2] + -12.387;
   1:L PR[91] R[100]mm/sec CNT100;
   1:  PR[91,1] = PR[90,1] + 87.928;
   1:  PR[91,2] = PR[90,2] + -11.623;
   1:L PR[91] R[100]mm/sec CNT100;
   1:  PR[91,1] = PR[90,1] + 89.669;
   1:  PR[91,2] = PR[90,2] + -8.826;
   1:L PR[91] R[100]mm/sec CNT100;
   1:  PR[91,1] = PR[90,1] + 91.047;
   1:  PR[91,2] = PR[90,2] + -4.872;
   1:L PR[91] R[100]mm/sec CNT100;
   1:  PR[91,1] = PR[90,1] + 91.193;
   1:  PR[91,2] = PR[90,2] + -3.604;
   1:L PR[91] R[100]mm/sec CNT100;
   1:  PR[91,1] = PR[90,1] + 91.572;
   1:  PR[91,2] = PR[90,2] + -1.114;
   1:L PR[91] R[100]mm/sec CNT100;
   1:  PR[91,1] = PR[90,1] + 91.607;
   1:  PR[91,2] = PR[90,2] + -0.801;
   1:L PR[91] R[100]mm/sec CNT100;
   1:  PR[91,1] = PR[90,1] + 91.372;
   1:  PR[91,2] = PR[90,2] + 0.468;
   1:L PR[91] R[100]mm/sec CNT100;
   1:  PR[91,1] = PR[90,1] + 91.045;
   1:  PR[91,2] = PR[90,2] + 3.417;
   1:L PR[91] R[100]mm/sec CNT100TB   .50sec,CALL END_PUD;
   1:  PR[92] = PR[91];
   1:  PR[92,3] = PR[92,3] + 20;
   1:J PR[92] 10% FINE;
   1:  PR[91,1] = PR[90,1] + 24.459;
   1:  PR[91,2] = PR[90,2] + -19.805;
   1:  PR[92] = PR[91];
   1:  PR[92,3] = PR[92,3] + 20;
   1:J PR[92] 10% FINE;
   1:L PR[91] R[100]mm/sec CNT100;
   1:  CALL LASER_DRAHT_START;
   1:  PR[91,1] = PR[90,1] + 29.392;
   1:  PR[91,2] = PR[90,2] + -19.144;
   1:L PR[91] R[100]mm/sec CNT100;
   1:  PR[91,1] = PR[90,1] + 33.986;
   1:  PR[91,2] = PR[90,2] + -17.234;
   1:L PR[91] R[100]mm/sec CNT100;
   1:  PR[91,1] = PR[90,1] + 34.996;
   1:  PR[91,2] = PR[90,2] + -16.469;
   1:L PR[91] R[100]mm/sec CNT100;
   1:  PR[91,1] = PR[90,1] + 37.921;
   1:  PR[91,2] = PR[90,2] + -14.213;
   1:L PR[91] R[100]mm/sec CNT100;
   1:  PR[91,1] = PR[90,1] + 38.674;
   1:  PR[91,2] = PR[90,2] + -13.250;
   1:L PR[91] R[100]mm/sec CNT100;
   1:  PR[91,1] = PR[90,1] + 41.002;
   1:  PR[91,2] = PR[90,2] + -10.202;
   1:L PR[91] R[100]mm/sec CNT100;
   1:  PR[91,1] = PR[90,1] + 41.006;
   1:  PR[91,2] = PR[90,2] + -10.195;
   1:L PR[91] R[100]mm/sec CNT100;
   1:  PR[91,1] = PR[90,1] + 42.478;
   1:  PR[91,2] = PR[90,2] + -6.631;
   1:L PR[91] R[100]mm/sec CNT100;
   1:  PR[91,1] = PR[90,1] + 42.735;
   1:  PR[91,2] = PR[90,2] + -6.057;
   1:L PR[91] R[100]mm/sec CNT100;
   1:  PR[91,1] = PR[90,1] + 42.992;
   1:  PR[91,2] = PR[90,2] + -5.050;
   1:L PR[91] R[100]mm/sec CNT100;
   1:  PR[91,1] = PR[90,1] + 43.381;
   1:  PR[91,2] = PR[90,2] + -2.091;
   1:L PR[91] R[100]mm/sec CNT100;
   1:  PR[91,1] = PR[90,1] + 43.498;
   1:  PR[91,2] = PR[90,2] + -0.772;
   1:L PR[91] R[100]mm/sec CNT100;
   1:  PR[91,1] = PR[90,1] + 43.139;
   1:  PR[91,2] = PR[90,2] + 1.951;
   1:L PR[91] R[100]mm/sec CNT100;
   1:  PR[91,1] = PR[90,1] + 42.991;
   1:  PR[91,2] = PR[90,2] + 3.577;
   1:L PR[91] R[100]mm/sec CNT100;
   1:  PR[91,1] = PR[90,1] + 42.700;
   1:  PR[91,2] = PR[90,2] + 4.702;
   1:L PR[91] R[100]mm/sec CNT100;
   1:  PR[91,1] = PR[90,1] + 41.393;
   1:  PR[91,2] = PR[90,2] + 7.870;
   1:L PR[91] R[100]mm/sec CNT100;
   1:  PR[91,1] = PR[90,1] + 41.029;
   1:  PR[91,2] = PR[90,2] + 8.694;
   1:L PR[91] R[100]mm/sec CNT100;
   1:  PR[91,1] = PR[90,1] + 41.002;
   1:  PR[91,2] = PR[90,2] + 8.744;
   1:L PR[91] R[100]mm/sec CNT100;
   1:  PR[91,1] = PR[90,1] + 38.663;
   1:  PR[91,2] = PR[90,2] + 11.810;
   1:L PR[91] R[100]mm/sec CNT100;
   1:  PR[91,1] = PR[90,1] + 37.914;
   1:  PR[91,2] = PR[90,2] + 12.762;
   1:L PR[91] R[100]mm/sec CNT100;
   1:  PR[91,1] = PR[90,1] + 34.989;
   1:  PR[91,2] = PR[90,2] + 15.018;
   1:L PR[91] R[100]mm/sec CNT100;
   1:  PR[91,1] = PR[90,1] + 33.975;
   1:  PR[91,2] = PR[90,2] + 15.782;
   1:L PR[91] R[100]mm/sec CNT100;
   1:  PR[91,1] = PR[90,1] + 30.626;
   1:  PR[91,2] = PR[90,2] + 17.182;
   1:L PR[91] R[100]mm/sec CNT100;
   1:  PR[91,1] = PR[90,1] + 29.388;
   1:  PR[91,2] = PR[90,2] + 17.687;
   1:L PR[91] R[100]mm/sec CNT100;
   1:  PR[91,1] = PR[90,1] + 24.450;
   1:  PR[91,2] = PR[90,2] + 18.346;
   1:L PR[91] R[100]mm/sec CNT100;
   1:  PR[91,1] = PR[90,1] + 19.510;
   1:  PR[91,2] = PR[90,2] + 17.707;
   1:L PR[91] R[100]mm/sec CNT100;
   1:  PR[91,1] = PR[90,1] + 16.366;
   1:  PR[91,2] = PR[90,2] + 16.420;
   1:L PR[91] R[100]mm/sec CNT100;
   1:  PR[91,1] = PR[90,1] + 14.901;
   1:  PR[91,2] = PR[90,2] + 15.814;
   1:L PR[91] R[100]mm/sec CNT100;
   1:  PR[91,1] = PR[90,1] + 10.931;
   1:  PR[91,2] = PR[90,2] + 12.787;
   1:L PR[91] R[100]mm/sec CNT100;
   1:  PR[91,1] = PR[90,1] + 7.883;
   1:  PR[91,2] = PR[90,2] + 8.833;
   1:L PR[91] R[100]mm/sec CNT100;
   1:  PR[91,1] = PR[90,1] + 6.643;
   1:  PR[91,2] = PR[90,2] + 5.854;
   1:L PR[91] R[100]mm/sec CNT100;
   1:  PR[91,1] = PR[90,1] + 5.965;
   1:  PR[91,2] = PR[90,2] + 4.223;
   1:L PR[91] R[100]mm/sec CNT100;
   1:  PR[91,1] = PR[90,1] + 5.310;
   1:  PR[91,2] = PR[90,2] + -0.729;
   1:L PR[91] R[100]mm/sec CNT100;
   1:  PR[91,1] = PR[90,1] + 5.965;
   1:  PR[91,2] = PR[90,2] + -5.683;
   1:L PR[91] R[100]mm/sec CNT100;
   1:  PR[91,1] = PR[90,1] + 7.885;
   1:  PR[91,2] = PR[90,2] + -10.295;
   1:L PR[91] R[100]mm/sec CNT100;
   1:  PR[91,1] = PR[90,1] + 8.936;
   1:  PR[91,2] = PR[90,2] + -11.660;
   1:L PR[91] R[100]mm/sec CNT100;
   1:  PR[91,1] = PR[90,1] + 10.935;
   1:  PR[91,2] = PR[90,2] + -14.249;
   1:L PR[91] R[100]mm/sec CNT100;
   1:  PR[91,1] = PR[90,1] + 14.905;
   1:  PR[91,2] = PR[90,2] + -17.275;
   1:L PR[91] R[100]mm/sec CNT100;
   1:  PR[91,1] = PR[90,1] + 19.521;
   1:  PR[91,2] = PR[90,2] + -19.169;
   1:L PR[91] R[100]mm/sec CNT100;
   1:  PR[91,1] = PR[90,1] + 21.012;
   1:  PR[91,2] = PR[90,2] + -19.365;
   1:L PR[91] R[100]mm/sec CNT100;
   1:  PR[91,1] = PR[90,1] + 24.459;
   1:  PR[91,2] = PR[90,2] + -19.805;
   1:L PR[91] R[100]mm/sec CNT100TB   .50sec,CALL END_PUD;
   1:  PR[92] = PR[91];
   1:  PR[92,3] = PR[92,3] + 20;
   1:J PR[92] 10% FINE;
   1:  PR[91,1] = PR[90,1] + -12.346;
   1:  PR[91,2] = PR[90,2] + 14.551;
   1:  PR[92] = PR[91];
   1:  PR[92,3] = PR[92,3] + 20;
   1:J PR[92] 10% FINE;
   1:L PR[91] R[100]mm/sec CNT100;
   1:  CALL LASER_DRAHT_START;
   1:  PR[91,1] = PR[90,1] + -15.179;
   1:  PR[91,2] = PR[90,2] + 16.250;
   1:L PR[91] R[100]mm/sec CNT100;
   1:  PR[91,1] = PR[90,1] + -19.233;
   1:  PR[91,2] = PR[90,2] + 17.587;
   1:L PR[91] R[100]mm/sec CNT100;
   1:  PR[91,1] = PR[90,1] + -20.779;
   1:  PR[91,2] = PR[90,2] + 17.747;
   1:L PR[91] R[100]mm/sec CNT100;
   1:  PR[91,1] = PR[90,1] + -23.460;
   1:  PR[91,2] = PR[90,2] + 17.998;
   1:L PR[91] R[100]mm/sec CNT100;
   1:  PR[91,1] = PR[90,1] + -25.292;
   1:  PR[91,2] = PR[90,2] + 17.779;
   1:L PR[91] R[100]mm/sec CNT100;
   1:  PR[91,1] = PR[90,1] + -27.663;
   1:  PR[91,2] = PR[90,2] + 17.472;
   1:L PR[91] R[100]mm/sec CNT100;
   1:  PR[91,1] = PR[90,1] + -29.647;
   1:  PR[91,2] = PR[90,2] + 16.769;
   1:L PR[91] R[100]mm/sec CNT100;
   1:  PR[91,1] = PR[90,1] + -31.633;
   1:  PR[91,2] = PR[90,2] + 16.046;
   1:L PR[91] R[100]mm/sec CNT100;
   1:  PR[91,1] = PR[90,1] + -33.599;
   1:  PR[91,2] = PR[90,2] + 14.805;
   1:L PR[91] R[100]mm/sec CNT100;
   1:  PR[91,1] = PR[90,1] + -35.174;
   1:  PR[91,2] = PR[90,2] + 13.794;
   1:L PR[91] R[100]mm/sec CNT100;
   1:  PR[91,1] = PR[90,1] + -38.124;
   1:  PR[91,2] = PR[90,2] + 10.827;
   1:L PR[91] R[100]mm/sec CNT100;
   1:  PR[91,1] = PR[90,1] + -40.335;
   1:  PR[91,2] = PR[90,2] + 7.301;
   1:L PR[91] R[100]mm/sec CNT100;
   1:  PR[91,1] = PR[90,1] + -41.703;
   1:  PR[91,2] = PR[90,2] + 3.385;
   1:L PR[91] R[100]mm/sec CNT100;
   1:  PR[91,1] = PR[90,1] + -42.024;
   1:  PR[91,2] = PR[90,2] + 0.555;
   1:L PR[91] R[100]mm/sec CNT100;
   1:  PR[91,1] = PR[90,1] + -42.096;
   1:  PR[91,2] = PR[90,2] + 0.206;
   1:L PR[91] R[100]mm/sec CNT100;
   1:  PR[91,1] = PR[90,1] + -42.199;
   1:  PR[91,2] = PR[90,2] + -0.717;
   1:L PR[91] R[100]mm/sec CNT100;
   1:  PR[91,1] = PR[90,1] + -41.858;
   1:  PR[91,2] = PR[90,2] + -3.458;
   1:L PR[91] R[100]mm/sec CNT100;
   1:  PR[91,1] = PR[90,1] + -41.703;
   1:  PR[91,2] = PR[90,2] + -4.845;
   1:L PR[91] R[100]mm/sec CNT100;
   1:  PR[91,1] = PR[90,1] + -40.335;
   1:  PR[91,2] = PR[90,2] + -8.760;
   1:L PR[91] R[100]mm/sec CNT100;
   1:  PR[91,1] = PR[90,1] + -38.124;
   1:  PR[91,2] = PR[90,2] + -12.286;
   1:L PR[91] R[100]mm/sec CNT100;
   1:  PR[91,1] = PR[90,1] + -35.177;
   1:  PR[91,2] = PR[90,2] + -15.250;
   1:L PR[91] R[100]mm/sec CNT100;
   1:  PR[91,1] = PR[90,1] + -31.637;
   1:  PR[91,2] = PR[90,2] + -17.501;
   1:L PR[91] R[100]mm/sec CNT100;
   1:  PR[91,1] = PR[90,1] + -29.583;
   1:  PR[91,2] = PR[90,2] + -18.228;
   1:L PR[91] R[100]mm/sec CNT100;
   1:  PR[91,1] = PR[90,1] + -27.663;
   1:  PR[91,2] = PR[90,2] + -18.928;
   1:L PR[91] R[100]mm/sec CNT100;
   1:  PR[91,1] = PR[90,1] + -25.725;
   1:  PR[91,2] = PR[90,2] + -19.160;
   1:L PR[91] R[100]mm/sec CNT100;
   1:  PR[91,1] = PR[90,1] + -23.460;
   1:  PR[91,2] = PR[90,2] + -19.455;
   1:L PR[91] R[100]mm/sec CNT100;
   1:  PR[91,1] = PR[90,1] + -21.772;
   1:  PR[91,2] = PR[90,2] + -19.279;
   1:L PR[91] R[100]mm/sec CNT100;
   1:  PR[91,1] = PR[90,1] + -19.230;
   1:  PR[91,2] = PR[90,2] + -19.043;
   1:L PR[91] R[100]mm/sec CNT100;
   1:  PR[91,1] = PR[90,1] + -17.879;
   1:  PR[91,2] = PR[90,2] + -18.587;
   1:L PR[91] R[100]mm/sec CNT100;
   1:  PR[91,1] = PR[90,1] + -15.178;
   1:  PR[91,2] = PR[90,2] + -17.708;
   1:L PR[91] R[100]mm/sec CNT100;
   1:  PR[91,1] = PR[90,1] + -11.528;
   1:  PR[91,2] = PR[90,2] + -15.508;
   1:L PR[91] R[100]mm/sec CNT100;
   1:  PR[91,1] = PR[90,1] + -8.458;
   1:  PR[91,2] = PR[90,2] + -12.546;
   1:L PR[91] R[100]mm/sec CNT100;
   1:  PR[91,1] = PR[90,1] + -6.135;
   1:  PR[91,2] = PR[90,2] + -8.970;
   1:L PR[91] R[100]mm/sec CNT100;
   1:  PR[91,1] = PR[90,1] + -4.693;
   1:  PR[91,2] = PR[90,2] + -4.972;
   1:L PR[91] R[100]mm/sec CNT100;
   1:  PR[91,1] = PR[90,1] + -4.248;
   1:  PR[91,2] = PR[90,2] + -0.740;
   1:L PR[91] R[100]mm/sec CNT100;
   1:  PR[91,1] = PR[90,1] + -4.260;
   1:  PR[91,2] = PR[90,2] + -0.638;
   1:L PR[91] R[100]mm/sec CNT100;
   1:  PR[91,1] = PR[90,1] + -4.247;
   1:  PR[91,2] = PR[90,2] + -0.309;
   1:L PR[91] R[100]mm/sec CNT100;
   1:  PR[91,1] = PR[90,1] + -4.689;
   1:  PR[91,2] = PR[90,2] + 3.503;
   1:L PR[91] R[100]mm/sec CNT100;
   1:  PR[91,1] = PR[90,1] + -6.135;
   1:  PR[91,2] = PR[90,2] + 7.511;
   1:L PR[91] R[100]mm/sec CNT100;
   1:  PR[91,1] = PR[90,1] + -8.458;
   1:  PR[91,2] = PR[90,2] + 11.087;
   1:L PR[91] R[100]mm/sec CNT100;
   1:  PR[91,1] = PR[90,1] + -11.533;
   1:  PR[91,2] = PR[90,2] + 14.054;
   1:L PR[91] R[100]mm/sec CNT100;
   1:  PR[91,1] = PR[90,1] + -12.346;
   1:  PR[91,2] = PR[90,2] + 14.551;
   1:L PR[91] R[100]mm/sec CNT100TB   .50sec,CALL END_PUD;
   1:  PR[92] = PR[91];
   1:  PR[92,3] = PR[92,3] + 20;
   1:J PR[92] 10% FINE;
   1:  PR[91,1] = PR[90,1] + -53.021;
   1:  PR[91,2] = PR[90,2] + -4.699;
   1:  PR[92] = PR[91];
   1:  PR[92,3] = PR[92,3] + 20;
   1:J PR[92] 10% FINE;
   1:L PR[91] R[100]mm/sec CNT100;
   1:  CALL LASER_DRAHT_START;
   1:  PR[91,1] = PR[90,1] + -52.877;
   1:  PR[91,2] = PR[90,2] + -3.452;
   1:L PR[91] R[100]mm/sec CNT100;
   1:  PR[91,1] = PR[90,1] + -52.683;
   1:  PR[91,2] = PR[90,2] + -0.769;
   1:L PR[91] R[100]mm/sec CNT100;
   1:  PR[91,1] = PR[90,1] + -53.132;
   1:  PR[91,2] = PR[90,2] + 3.242;
   1:L PR[91] R[100]mm/sec CNT100;
   1:  PR[91,1] = PR[90,1] + -54.462;
   1:  PR[91,2] = PR[90,2] + 7.021;
   1:L PR[91] R[100]mm/sec CNT100;
   1:  PR[91,1] = PR[90,1] + -56.604;
   1:  PR[91,2] = PR[90,2] + 10.437;
   1:L PR[91] R[100]mm/sec CNT100;
   1:  PR[91,1] = PR[90,1] + -59.447;
   1:  PR[91,2] = PR[90,2] + 13.338;
   1:L PR[91] R[100]mm/sec CNT100;
   1:  PR[91,1] = PR[90,1] + -60.836;
   1:  PR[91,2] = PR[90,2] + 14.269;
   1:L PR[91] R[100]mm/sec CNT100;
   1:  PR[91,1] = PR[90,1] + -62.844;
   1:  PR[91,2] = PR[90,2] + 15.588;
   1:L PR[91] R[100]mm/sec CNT100;
   1:  PR[91,1] = PR[90,1] + -65.077;
   1:  PR[91,2] = PR[90,2] + 16.491;
   1:L PR[91] R[100]mm/sec CNT100;
   1:  PR[91,1] = PR[90,1] + -66.638;
   1:  PR[91,2] = PR[90,2] + 17.105;
   1:L PR[91] R[100]mm/sec CNT100;
   1:  PR[91,1] = PR[90,1] + -70.671;
   1:  PR[91,2] = PR[90,2] + 17.834;
   1:L PR[91] R[100]mm/sec CNT100;
   1:  PR[91,1] = PR[90,1] + -74.749;
   1:  PR[91,2] = PR[90,2] + 17.750;
   1:L PR[91] R[100]mm/sec CNT100;
   1:  PR[91,1] = PR[90,1] + -78.684;
   1:  PR[91,2] = PR[90,2] + 16.871;
   1:L PR[91] R[100]mm/sec CNT100;
   1:  PR[91,1] = PR[90,1] + -82.248;
   1:  PR[91,2] = PR[90,2] + 15.256;
   1:L PR[91] R[100]mm/sec CNT100;
   1:  PR[91,1] = PR[90,1] + -85.392;
   1:  PR[91,2] = PR[90,2] + 12.958;
   1:L PR[91] R[100]mm/sec CNT100;
   1:  PR[91,1] = PR[90,1] + -87.981;
   1:  PR[91,2] = PR[90,2] + 10.077;
   1:L PR[91] R[100]mm/sec CNT100;
   1:  PR[91,1] = PR[90,1] + -89.911;
   1:  PR[91,2] = PR[90,2] + 6.739;
   1:L PR[91] R[100]mm/sec CNT100;
   1:  PR[91,1] = PR[90,1] + -91.101;
   1:  PR[91,2] = PR[90,2] + 3.084;
   1:L PR[91] R[100]mm/sec CNT100;
   1:  PR[91,1] = PR[90,1] + -91.213;
   1:  PR[91,2] = PR[90,2] + 2.037;
   1:L PR[91] R[100]mm/sec CNT100;
   1:  PR[91,1] = PR[90,1] + -91.473;
   1:  PR[91,2] = PR[90,2] + 0.383;
   1:L PR[91] R[100]mm/sec CNT100;
   1:  PR[91,1] = PR[90,1] + -91.586;
   1:  PR[91,2] = PR[90,2] + -0.678;
   1:L PR[91] R[100]mm/sec CNT100;
   1:  PR[91,1] = PR[90,1] + -91.419;
   1:  PR[91,2] = PR[90,2] + -1.736;
   1:L PR[91] R[100]mm/sec CNT100;
   1:  PR[91,1] = PR[90,1] + -91.277;
   1:  PR[91,2] = PR[90,2] + -2.342;
   1:L PR[91] R[100]mm/sec CNT100;
   1:  PR[91,1] = PR[90,1] + -91.046;
   1:  PR[91,2] = PR[90,2] + -4.545;
   1:L PR[91] R[100]mm/sec CNT100;
   1:  PR[91,1] = PR[90,1] + -90.520;
   1:  PR[91,2] = PR[90,2] + -6.151;
   1:L PR[91] R[100]mm/sec CNT100;
   1:  PR[91,1] = PR[90,1] + -89.854;
   1:  PR[91,2] = PR[90,2] + -8.202;
   1:L PR[91] R[100]mm/sec CNT100;
   1:  PR[91,1] = PR[90,1] + -87.918;
   1:  PR[91,2] = PR[90,2] + -11.542;
   1:L PR[91] R[100]mm/sec CNT100;
   1:  PR[91,1] = PR[90,1] + -85.320;
   1:  PR[91,2] = PR[90,2] + -14.427;
   1:L PR[91] R[100]mm/sec CNT100;
   1:  PR[91,1] = PR[90,1] + -82.165;
   1:  PR[91,2] = PR[90,2] + -16.729;
   1:L PR[91] R[100]mm/sec CNT100;
   1:  PR[91,1] = PR[90,1] + -78.585;
   1:  PR[91,2] = PR[90,2] + -18.350;
   1:L PR[91] R[100]mm/sec CNT100;
   1:  PR[91,1] = PR[90,1] + -74.729;
   1:  PR[91,2] = PR[90,2] + -19.214;
   1:L PR[91] R[100]mm/sec CNT100;
   1:  PR[91,1] = PR[90,1] + -70.750;
   1:  PR[91,2] = PR[90,2] + -19.278;
   1:L PR[91] R[100]mm/sec CNT100;
   1:  PR[91,1] = PR[90,1] + -66.695;
   1:  PR[91,2] = PR[90,2] + -18.552;
   1:L PR[91] R[100]mm/sec CNT100;
   1:  PR[91,1] = PR[90,1] + -63.514;
   1:  PR[91,2] = PR[90,2] + -17.287;
   1:L PR[91] R[100]mm/sec CNT100;
   1:  PR[91,1] = PR[90,1] + -62.844;
   1:  PR[91,2] = PR[90,2] + -17.032;
   1:L PR[91] R[100]mm/sec CNT100;
   1:  PR[91,1] = PR[90,1] + -60.434;
   1:  PR[91,2] = PR[90,2] + -15.440;
   1:L PR[91] R[100]mm/sec CNT100;
   1:  PR[91,1] = PR[90,1] + -59.408;
   1:  PR[91,2] = PR[90,2] + -14.784;
   1:L PR[91] R[100]mm/sec CNT100;
   1:  PR[91,1] = PR[90,1] + -57.744;
   1:  PR[91,2] = PR[90,2] + -13.089;
   1:L PR[91] R[100]mm/sec CNT100;
   1:  PR[91,1] = PR[90,1] + -56.537;
   1:  PR[91,2] = PR[90,2] + -11.891;
   1:L PR[91] R[100]mm/sec CNT100;
   1:  PR[91,1] = PR[90,1] + -55.519;
   1:  PR[91,2] = PR[90,2] + -10.270;
   1:L PR[91] R[100]mm/sec CNT100;
   1:  PR[91,1] = PR[90,1] + -54.367;
   1:  PR[91,2] = PR[90,2] + -8.475;
   1:L PR[91] R[100]mm/sec CNT100;
   1:  PR[91,1] = PR[90,1] + -53.021;
   1:  PR[91,2] = PR[90,2] + -4.699;
   1:L PR[91] R[100]mm/sec CNT100TB   .50sec,CALL END_PUD;
   1:  PR[92] = PR[91];
   1:  PR[92,3] = PR[92,3] + 20;
   1:J PR[92] 10% FINE;
   1:  PR[91] = PR[90];
   1:  PR[91,1] = PR[90,1] + 87.268;
   1:  PR[91,2] = PR[90,2] + -12.439;
   1:  PR[91,3] = PR[90,3] + 28.795;
   1:  PR[92] = PR[91];
   1:  PR[92,3] = PR[92,3] + 20;
   1:J PR[92] 10% FINE;
   1:L PR[91] R[100]mm/sec CNT100;
   1:  CALL LASER_DRAHT_START;
   1:  PR[91,1] = PR[90,1] + 89.501;
   1:  PR[91,2] = PR[90,2] + -8.857;
   1:L PR[91] R[100]mm/sec CNT100;
   1:  PR[91,1] = PR[90,1] + 90.883;
   1:  PR[91,2] = PR[90,2] + -4.888;
   1:L PR[91] R[100]mm/sec CNT100;
   1:  PR[91,1] = PR[90,1] + 90.967;
   1:  PR[91,2] = PR[90,2] + -4.156;
   1:L PR[91] R[100]mm/sec CNT100;
   1:  PR[91,1] = PR[90,1] + 91.206;
   1:  PR[91,2] = PR[90,2] + -2.585;
   1:L PR[91] R[100]mm/sec CNT100;
   1:  PR[91,1] = PR[90,1] + 91.407;
   1:  PR[91,2] = PR[90,2] + -0.801;
   1:L PR[91] R[100]mm/sec CNT100;
   1:  PR[91,1] = PR[90,1] + 91.267;
   1:  PR[91,2] = PR[90,2] + -0.043;
   1:L PR[91] R[100]mm/sec CNT100;
   1:  PR[91,1] = PR[90,1] + 90.881;
   1:  PR[91,2] = PR[90,2] + 3.433;
   1:L PR[91] R[100]mm/sec CNT100;
   1:  PR[91,1] = PR[90,1] + 89.501;
   1:  PR[91,2] = PR[90,2] + 7.398;
   1:L PR[91] R[100]mm/sec CNT100;
   1:  PR[91,1] = PR[90,1] + 87.268;
   1:  PR[91,2] = PR[90,2] + 10.980;
   1:L PR[91] R[100]mm/sec CNT100;
   1:  PR[91,1] = PR[90,1] + 84.286;
   1:  PR[91,2] = PR[90,2] + 14.005;
   1:L PR[91] R[100]mm/sec CNT100;
   1:  PR[91,1] = PR[90,1] + 80.640;
   1:  PR[91,2] = PR[90,2] + 16.343;
   1:L PR[91] R[100]mm/sec CNT100;
   1:  PR[91,1] = PR[90,1] + 76.908;
   1:  PR[91,2] = PR[90,2] + 17.710;
   1:L PR[91] R[100]mm/sec CNT100;
   1:  PR[91,1] = PR[90,1] + 76.441;
   1:  PR[91,2] = PR[90,2] + 17.891;
   1:L PR[91] R[100]mm/sec CNT100;
   1:  PR[91,1] = PR[90,1] + 73.048;
   1:  PR[91,2] = PR[90,2] + 18.366;
   1:L PR[91] R[100]mm/sec CNT100;
   1:  PR[91,1] = PR[90,1] + 71.961;
   1:  PR[91,2] = PR[90,2] + 18.540;
   1:L PR[91] R[100]mm/sec CNT100;
   1:  PR[91,1] = PR[90,1] + 69.180;
   1:  PR[91,2] = PR[90,2] + 18.333;
   1:L PR[91] R[100]mm/sec CNT100;
   1:  PR[91,1] = PR[90,1] + 67.396;
   1:  PR[91,2] = PR[90,2] + 18.240;
   1:L PR[91] R[100]mm/sec CNT100;
   1:  PR[91,1] = PR[90,1] + 65.418;
   1:  PR[91,2] = PR[90,2] + 17.653;
   1:L PR[91] R[100]mm/sec CNT100;
   1:  PR[91,1] = PR[90,1] + 62.965;
   1:  PR[91,2] = PR[90,2] + 16.985;
   1:L PR[91] R[100]mm/sec CNT100;
   1:  PR[91,1] = PR[90,1] + 61.856;
   1:  PR[91,2] = PR[90,2] + 16.368;
   1:L PR[91] R[100]mm/sec CNT100;
   1:  PR[91,1] = PR[90,1] + 58.893;
   1:  PR[91,2] = PR[90,2] + 14.805;
   1:L PR[91] R[100]mm/sec CNT100;
   1:  PR[91,1] = PR[90,1] + 58.565;
   1:  PR[91,2] = PR[90,2] + 14.510;
   1:L PR[91] R[100]mm/sec CNT100;
   1:  PR[91,1] = PR[90,1] + 55.784;
   1:  PR[91,2] = PR[90,2] + 12.108;
   1:L PR[91] R[100]mm/sec CNT100;
   1:  PR[91,1] = PR[90,1] + 55.300;
   1:  PR[91,2] = PR[90,2] + 11.720;
   1:L PR[91] R[100]mm/sec CNT100;
   1:  PR[91,1] = PR[90,1] + 52.540;
   1:  PR[91,2] = PR[90,2] + 8.136;
   1:L PR[91] R[100]mm/sec CNT100;
   1:  PR[91,1] = PR[90,1] + 52.071;
   1:  PR[91,2] = PR[90,2] + 7.140;
   1:L PR[91] R[100]mm/sec CNT100;
   1:  PR[91,1] = PR[90,1] + 50.705;
   1:  PR[91,2] = PR[90,2] + 3.916;
   1:L PR[91] R[100]mm/sec CNT100;
   1:  PR[91,1] = PR[90,1] + 50.446;
   1:  PR[91,2] = PR[90,2] + 2.223;
   1:L PR[91] R[100]mm/sec CNT100;
   1:  PR[91,1] = PR[90,1] + 50.038;
   1:  PR[91,2] = PR[90,2] + -0.729;
   1:L PR[91] R[100]mm/sec CNT100;
   1:  PR[91,1] = PR[90,1] + 50.446;
   1:  PR[91,2] = PR[90,2] + -3.684;
   1:L PR[91] R[100]mm/sec CNT100;
   1:  PR[91,1] = PR[90,1] + 50.704;
   1:  PR[91,2] = PR[90,2] + -5.374;
   1:L PR[91] R[100]mm/sec CNT100;
   1:  PR[91,1] = PR[90,1] + 52.071;
   1:  PR[91,2] = PR[90,2] + -8.598;
   1:L PR[91] R[100]mm/sec CNT100;
   1:  PR[91,1] = PR[90,1] + 52.540;
   1:  PR[91,2] = PR[90,2] + -9.595;
   1:L PR[91] R[100]mm/sec CNT100;
   1:  PR[91,1] = PR[90,1] + 55.300;
   1:  PR[91,2] = PR[90,2] + -13.179;
   1:L PR[91] R[100]mm/sec CNT100;
   1:  PR[91,1] = PR[90,1] + 55.787;
   1:  PR[91,2] = PR[90,2] + -13.569;
   1:L PR[91] R[100]mm/sec CNT100;
   1:  PR[91,1] = PR[90,1] + 58.893;
   1:  PR[91,2] = PR[90,2] + -16.268;
   1:L PR[91] R[100]mm/sec CNT100;
   1:  PR[91,1] = PR[90,1] + 59.466;
   1:  PR[91,2] = PR[90,2] + -16.585;
   1:L PR[91] R[100]mm/sec CNT100;
   1:  PR[91,1] = PR[90,1] + 62.965;
   1:  PR[91,2] = PR[90,2] + -18.448;
   1:L PR[91] R[100]mm/sec CNT100;
   1:  PR[91,1] = PR[90,1] + 64.665;
   1:  PR[91,2] = PR[90,2] + -18.947;
   1:L PR[91] R[100]mm/sec CNT100;
   1:  PR[91,1] = PR[90,1] + 67.396;
   1:  PR[91,2] = PR[90,2] + -19.702;
   1:L PR[91] R[100]mm/sec CNT100;
   1:  PR[91,1] = PR[90,1] + 70.206;
   1:  PR[91,2] = PR[90,2] + -19.904;
   1:L PR[91] R[100]mm/sec CNT100;
   1:  PR[91,1] = PR[90,1] + 71.961;
   1:  PR[91,2] = PR[90,2] + -20.003;
   1:L PR[91] R[100]mm/sec CNT100;
   1:  PR[91,1] = PR[90,1] + 75.629;
   1:  PR[91,2] = PR[90,2] + -19.481;
   1:L PR[91] R[100]mm/sec CNT100;
   1:  PR[91,1] = PR[90,1] + 76.441;
   1:  PR[91,2] = PR[90,2] + -19.353;
   1:L PR[91] R[100]mm/sec CNT100;
   1:  PR[91,1] = PR[90,1] + 80.638;
   1:  PR[91,2] = PR[90,2] + -17.803;
   1:L PR[91] R[100]mm/sec CNT100;
   1:  PR[91,1] = PR[90,1] + 84.286;
   1:  PR[91,2] = PR[90,2] + -15.464;
   1:L PR[91] R[100]mm/sec CNT100;
   1:  PR[91,1] = PR[90,1] + 87.268;
   1:  PR[91,2] = PR[90,2] + -12.439;
   1:L PR[91] R[100]mm/sec CNT100TB   .50sec,CALL END_PUD;
   1:  PR[92] = PR[91];
   1:  PR[92,3] = PR[92,3] + 20;
   1:J PR[92] 10% FINE;
   1:  PR[91,1] = PR[90,1] + 39.000;
   1:  PR[91,2] = PR[90,2] + -12.973;
   1:  PR[92] = PR[91];
   1:  PR[92,3] = PR[92,3] + 20;
   1:J PR[92] 10% FINE;
   1:L PR[91] R[100]mm/sec CNT100;
   1:  CALL LASER_DRAHT_START;
   1:  PR[91,1] = PR[90,1] + 41.047;
   1:  PR[91,2] = PR[90,2] + -10.293;
   1:L PR[91] R[100]mm/sec CNT100;
   1:  PR[91,1] = PR[90,1] + 41.096;
   1:  PR[91,2] = PR[90,2] + -10.205;
   1:L PR[91] R[100]mm/sec CNT100;
   1:  PR[91,1] = PR[90,1] + 42.376;
   1:  PR[91,2] = PR[90,2] + -7.104;
   1:L PR[91] R[100]mm/sec CNT100;
   1:  PR[91,1] = PR[90,1] + 42.743;
   1:  PR[91,2] = PR[90,2] + -6.285;
   1:L PR[91] R[100]mm/sec CNT100;
   1:  PR[91,1] = PR[90,1] + 43.114;
   1:  PR[91,2] = PR[90,2] + -4.830;
   1:L PR[91] R[100]mm/sec CNT100;
   1:  PR[91,1] = PR[90,1] + 43.402;
   1:  PR[91,2] = PR[90,2] + -2.639;
   1:L PR[91] R[100]mm/sec CNT100;
   1:  PR[91,1] = PR[90,1] + 43.567;
   1:  PR[91,2] = PR[90,2] + -0.772;
   1:L PR[91] R[100]mm/sec CNT100;
   1:  PR[91,1] = PR[90,1] + 43.320;
   1:  PR[91,2] = PR[90,2] + 1.105;
   1:L PR[91] R[100]mm/sec CNT100;
   1:  PR[91,1] = PR[90,1] + 43.117;
   1:  PR[91,2] = PR[90,2] + 3.338;
   1:L PR[91] R[100]mm/sec CNT100;
   1:  PR[91,1] = PR[90,1] + 42.699;
   1:  PR[91,2] = PR[90,2] + 4.957;
   1:L PR[91] R[100]mm/sec CNT100;
   1:  PR[91,1] = PR[90,1] + 41.626;
   1:  PR[91,2] = PR[90,2] + 7.556;
   1:L PR[91] R[100]mm/sec CNT100;
   1:  PR[91,1] = PR[90,1] + 41.123;
   1:  PR[91,2] = PR[90,2] + 8.695;
   1:L PR[91] R[100]mm/sec CNT100;
   1:  PR[91,1] = PR[90,1] + 41.047;
   1:  PR[91,2] = PR[90,2] + 8.834;
   1:L PR[91] R[100]mm/sec CNT100;
   1:  PR[91,1] = PR[90,1] + 38.984;
   1:  PR[91,2] = PR[90,2] + 11.540;
   1:L PR[91] R[100]mm/sec CNT100;
   1:  PR[91,1] = PR[90,1] + 37.931;
   1:  PR[91,2] = PR[90,2] + 12.880;
   1:L PR[91] R[100]mm/sec CNT100;
   1:  PR[91,1] = PR[90,1] + 35.373;
   1:  PR[91,2] = PR[90,2] + 14.853;
   1:L PR[91] R[100]mm/sec CNT100;
   1:  PR[91,1] = PR[90,1] + 33.963;
   1:  PR[91,2] = PR[90,2] + 15.915;
   1:L PR[91] R[100]mm/sec CNT100;
   1:  PR[91,1] = PR[90,1] + 31.045;
   1:  PR[91,2] = PR[90,2] + 17.135;
   1:L PR[91] R[100]mm/sec CNT100;
   1:  PR[91,1] = PR[90,1] + 29.344;
   1:  PR[91,2] = PR[90,2] + 17.828;
   1:L PR[91] R[100]mm/sec CNT100;
   1:  PR[91,1] = PR[90,1] + 24.373;
   1:  PR[91,2] = PR[90,2] + 18.489;
   1:L PR[91] R[100]mm/sec CNT100;
   1:  PR[91,1] = PR[90,1] + 19.398;
   1:  PR[91,2] = PR[90,2] + 17.843;
   1:L PR[91] R[100]mm/sec CNT100;
   1:  PR[91,1] = PR[90,1] + 16.701;
   1:  PR[91,2] = PR[90,2] + 16.739;
   1:L PR[91] R[100]mm/sec CNT100;
   1:  PR[91,1] = PR[90,1] + 14.758;
   1:  PR[91,2] = PR[90,2] + 15.935;
   1:L PR[91] R[100]mm/sec CNT100;
   1:  PR[91,1] = PR[90,1] + 10.760;
   1:  PR[91,2] = PR[90,2] + 12.885;
   1:L PR[91] R[100]mm/sec CNT100;
   1:  PR[91,1] = PR[90,1] + 7.691;
   1:  PR[91,2] = PR[90,2] + 8.902;
   1:L PR[91] R[100]mm/sec CNT100;
   1:  PR[91,1] = PR[90,1] + 6.643;
   1:  PR[91,2] = PR[90,2] + 6.385;
   1:L PR[91] R[100]mm/sec CNT100;
   1:  PR[91,1] = PR[90,1] + 5.759;
   1:  PR[91,2] = PR[90,2] + 4.259;
   1:L PR[91] R[100]mm/sec CNT100;
   1:  PR[91,1] = PR[90,1] + 5.100;
   1:  PR[91,2] = PR[90,2] + -0.729;
   1:L PR[91] R[100]mm/sec CNT100;
   1:  PR[91,1] = PR[90,1] + 5.760;
   1:  PR[91,2] = PR[90,2] + -5.720;
   1:L PR[91] R[100]mm/sec CNT100;
   1:  PR[91,1] = PR[90,1] + 7.694;
   1:  PR[91,2] = PR[90,2] + -10.366;
   1:L PR[91] R[100]mm/sec CNT100;
   1:  PR[91,1] = PR[90,1] + 9.071;
   1:  PR[91,2] = PR[90,2] + -12.153;
   1:L PR[91] R[100]mm/sec CNT100;
   1:  PR[91,1] = PR[90,1] + 10.765;
   1:  PR[91,2] = PR[90,2] + -14.349;
   1:L PR[91] R[100]mm/sec CNT100;
   1:  PR[91,1] = PR[90,1] + 14.764;
   1:  PR[91,2] = PR[90,2] + -17.397;
   1:L PR[91] R[100]mm/sec CNT100;
   1:  PR[91,1] = PR[90,1] + 19.412;
   1:  PR[91,2] = PR[90,2] + -19.306;
   1:L PR[91] R[100]mm/sec CNT100;
   1:  PR[91,1] = PR[90,1] + 21.410;
   1:  PR[91,2] = PR[90,2] + -19.568;
   1:L PR[91] R[100]mm/sec CNT100;
   1:  PR[91,1] = PR[90,1] + 24.384;
   1:  PR[91,2] = PR[90,2] + -19.948;
   1:L PR[91] R[100]mm/sec CNT100;
   1:  PR[91,1] = PR[90,1] + 29.352;
   1:  PR[91,2] = PR[90,2] + -19.284;
   1:L PR[91] R[100]mm/sec CNT100;
   1:  PR[91,1] = PR[90,1] + 33.978;
   1:  PR[91,2] = PR[90,2] + -17.364;
   1:L PR[91] R[100]mm/sec CNT100;
   1:  PR[91,1] = PR[90,1] + 35.384;
   1:  PR[91,2] = PR[90,2] + -16.300;
   1:L PR[91] R[100]mm/sec CNT100;
   1:  PR[91,1] = PR[90,1] + 37.942;
   1:  PR[91,2] = PR[90,2] + -14.327;
   1:L PR[91] R[100]mm/sec CNT100;
   1:  PR[91,1] = PR[90,1] + 39.000;
   1:  PR[91,2] = PR[90,2] + -12.973;
   1:L PR[91] R[100]mm/sec CNT100TB   .50sec,CALL END_PUD;
   1:  PR[92] = PR[91];
   1:  PR[92,3] = PR[92,3] + 20;
   1:J PR[92] 10% FINE;
   1:  PR[91,1] = PR[90,1] + -35.031;
   1:  PR[91,2] = PR[90,2] + -15.307;
   1:  PR[92] = PR[91];
   1:  PR[92,3] = PR[92,3] + 20;
   1:J PR[92] 10% FINE;
   1:L PR[91] R[100]mm/sec CNT100;
   1:  CALL LASER_DRAHT_START;
   1:  PR[91,1] = PR[90,1] + -31.479;
   1:  PR[91,2] = PR[90,2] + -17.570;
   1:L PR[91] R[100]mm/sec CNT100;
   1:  PR[91,1] = PR[90,1] + -29.846;
   1:  PR[91,2] = PR[90,2] + -18.148;
   1:L PR[91] R[100]mm/sec CNT100;
   1:  PR[91,1] = PR[90,1] + -27.490;
   1:  PR[91,2] = PR[90,2] + -19.008;
   1:L PR[91] R[100]mm/sec CNT100;
   1:  PR[91,1] = PR[90,1] + -26.011;
   1:  PR[91,2] = PR[90,2] + -19.184;
   1:L PR[91] R[100]mm/sec CNT100;
   1:  PR[91,1] = PR[90,1] + -23.269;
   1:  PR[91,2] = PR[90,2] + -19.541;
   1:L PR[91] R[100]mm/sec CNT100;
   1:  PR[91,1] = PR[90,1] + -22.057;
   1:  PR[91,2] = PR[90,2] + -19.415;
   1:L PR[91] R[100]mm/sec CNT100;
   1:  PR[91,1] = PR[90,1] + -19.010;
   1:  PR[91,2] = PR[90,2] + -19.132;
   1:L PR[91] R[100]mm/sec CNT100;
   1:  PR[91,1] = PR[90,1] + -14.945;
   1:  PR[91,2] = PR[90,2] + -17.797;
   1:L PR[91] R[100]mm/sec CNT100;
   1:  PR[91,1] = PR[90,1] + -11.270;
   1:  PR[91,2] = PR[90,2] + -15.588;
   1:L PR[91] R[100]mm/sec CNT100;
   1:  PR[91,1] = PR[90,1] + -8.180;
   1:  PR[91,2] = PR[90,2] + -12.612;
   1:L PR[91] R[100]mm/sec CNT100;
   1:  PR[91,1] = PR[90,1] + -5.841;
   1:  PR[91,2] = PR[90,2] + -9.017;
   1:L PR[91] R[100]mm/sec CNT100;
   1:  PR[91,1] = PR[90,1] + -4.786;
   1:  PR[91,2] = PR[90,2] + -6.096;
   1:L PR[91] R[100]mm/sec CNT100;
   1:  PR[91,1] = PR[90,1] + -4.371;
   1:  PR[91,2] = PR[90,2] + -4.985;
   1:L PR[91] R[100]mm/sec CNT100;
   1:  PR[91,1] = PR[90,1] + -3.858;
   1:  PR[91,2] = PR[90,2] + -0.763;
   1:L PR[91] R[100]mm/sec CNT100;
   1:  PR[91,1] = PR[90,1] + -4.364;
   1:  PR[91,2] = PR[90,2] + 3.490;
   1:L PR[91] R[100]mm/sec CNT100;
   1:  PR[91,1] = PR[90,1] + -5.841;
   1:  PR[91,2] = PR[90,2] + 7.557;
   1:L PR[91] R[100]mm/sec CNT100;
   1:  PR[91,1] = PR[90,1] + -8.180;
   1:  PR[91,2] = PR[90,2] + 11.154;
   1:L PR[91] R[100]mm/sec CNT100;
   1:  PR[91,1] = PR[90,1] + -11.276;
   1:  PR[91,2] = PR[90,2] + 14.134;
   1:L PR[91] R[100]mm/sec CNT100;
   1:  PR[91,1] = PR[90,1] + -11.596;
   1:  PR[91,2] = PR[90,2] + 14.330;
   1:L PR[91] R[100]mm/sec CNT100;
   1:  PR[91,1] = PR[90,1] + -14.944;
   1:  PR[91,2] = PR[90,2] + 16.337;
   1:L PR[91] R[100]mm/sec CNT100;
   1:  PR[91,1] = PR[90,1] + -19.013;
   1:  PR[91,2] = PR[90,2] + 17.674;
   1:L PR[91] R[100]mm/sec CNT100;
   1:  PR[91,1] = PR[90,1] + -23.265;
   1:  PR[91,2] = PR[90,2] + 18.084;
   1:L PR[91] R[100]mm/sec CNT100;
   1:  PR[91,1] = PR[90,1] + -27.488;
   1:  PR[91,2] = PR[90,2] + 17.551;
   1:L PR[91] R[100]mm/sec CNT100;
   1:  PR[91,1] = PR[90,1] + -31.478;
   1:  PR[91,2] = PR[90,2] + 16.113;
   1:L PR[91] R[100]mm/sec CNT100;
   1:  PR[91,1] = PR[90,1] + -33.041;
   1:  PR[91,2] = PR[90,2] + 15.126;
   1:L PR[91] R[100]mm/sec CNT100;
   1:  PR[91,1] = PR[90,1] + -35.028;
   1:  PR[91,2] = PR[90,2] + 13.851;
   1:L PR[91] R[100]mm/sec CNT100;
   1:  PR[91,1] = PR[90,1] + -37.988;
   1:  PR[91,2] = PR[90,2] + 10.872;
   1:L PR[91] R[100]mm/sec CNT100;
   1:  PR[91,1] = PR[90,1] + -40.205;
   1:  PR[91,2] = PR[90,2] + 7.331;
   1:L PR[91] R[100]mm/sec CNT100;
   1:  PR[91,1] = PR[90,1] + -41.577;
   1:  PR[91,2] = PR[90,2] + 3.400;
   1:L PR[91] R[100]mm/sec CNT100;
   1:  PR[91,1] = PR[90,1] + -41.851;
   1:  PR[91,2] = PR[90,2] + 0.989;
   1:L PR[91] R[100]mm/sec CNT100;
   1:  PR[91,1] = PR[90,1] + -41.912;
   1:  PR[91,2] = PR[90,2] + 0.689;
   1:L PR[91] R[100]mm/sec CNT100;
   1:  PR[91,1] = PR[90,1] + -42.070;
   1:  PR[91,2] = PR[90,2] + -0.717;
   1:L PR[91] R[100]mm/sec CNT100;
   1:  PR[91,1] = PR[90,1] + -41.780;
   1:  PR[91,2] = PR[90,2] + -3.046;
   1:L PR[91] R[100]mm/sec CNT100;
   1:  PR[91,1] = PR[90,1] + -41.577;
   1:  PR[91,2] = PR[90,2] + -4.860;
   1:L PR[91] R[100]mm/sec CNT100;
   1:  PR[91,1] = PR[90,1] + -40.205;
   1:  PR[91,2] = PR[90,2] + -8.790;
   1:L PR[91] R[100]mm/sec CNT100;
   1:  PR[91,1] = PR[90,1] + -37.988;
   1:  PR[91,2] = PR[90,2] + -12.331;
   1:L PR[91] R[100]mm/sec CNT100;
   1:  PR[91,1] = PR[90,1] + -35.031;
   1:  PR[91,2] = PR[90,2] + -15.307;
   1:L PR[91] R[100]mm/sec CNT100TB   .50sec,CALL END_PUD;
   1:  PR[92] = PR[91];
   1:  PR[92,3] = PR[92,3] + 20;
   1:J PR[92] 10% FINE;
   1:  PR[91,1] = PR[90,1] + -52.444;
   1:  PR[91,2] = PR[90,2] + -4.731;
   1:  PR[92] = PR[91];
   1:  PR[92,3] = PR[92,3] + 20;
   1:J PR[92] 10% FINE;
   1:L PR[91] R[100]mm/sec CNT100;
   1:  CALL LASER_DRAHT_START;
   1:  PR[91,1] = PR[90,1] + -52.394;
   1:  PR[91,2] = PR[90,2] + -4.297;
   1:L PR[91] R[100]mm/sec CNT100;
   1:  PR[91,1] = PR[90,1] + -52.278;
   1:  PR[91,2] = PR[90,2] + -2.705;
   1:L PR[91] R[100]mm/sec CNT100;
   1:  PR[91,1] = PR[90,1] + -52.049;
   1:  PR[91,2] = PR[90,2] + -0.729;
   1:L PR[91] R[100]mm/sec CNT100;
   1:  PR[91,1] = PR[90,1] + -52.298;
   1:  PR[91,2] = PR[90,2] + 1.418;
   1:L PR[91] R[100]mm/sec CNT100;
   1:  PR[91,1] = PR[90,1] + -52.415;
   1:  PR[91,2] = PR[90,2] + 2.813;
   1:L PR[91] R[100]mm/sec CNT100;
   1:  PR[91,1] = PR[90,1] + -52.468;
   1:  PR[91,2] = PR[90,2] + 3.254;
   1:L PR[91] R[100]mm/sec CNT100;
   1:  PR[91,1] = PR[90,1] + -53.877;
   1:  PR[91,2] = PR[90,2] + 7.045;
   1:L PR[91] R[100]mm/sec CNT100;
   1:  PR[91,1] = PR[90,1] + -55.077;
   1:  PR[91,2] = PR[90,2] + 8.853;
   1:L PR[91] R[100]mm/sec CNT100;
   1:  PR[91,1] = PR[90,1] + -56.120;
   1:  PR[91,2] = PR[90,2] + 10.513;
   1:L PR[91] R[100]mm/sec CNT100;
   1:  PR[91,1] = PR[90,1] + -58.984;
   1:  PR[91,2] = PR[90,2] + 13.425;
   1:L PR[91] R[100]mm/sec CNT100;
   1:  PR[91,1] = PR[90,1] + -62.416;
   1:  PR[91,2] = PR[90,2] + 15.689;
   1:L PR[91] R[100]mm/sec CNT100;
   1:  PR[91,1] = PR[90,1] + -63.818;
   1:  PR[91,2] = PR[90,2] + 16.256;
   1:L PR[91] R[100]mm/sec CNT100;
   1:  PR[91,1] = PR[90,1] + -66.237;
   1:  PR[91,2] = PR[90,2] + 17.207;
   1:L PR[91] R[100]mm/sec CNT100;
   1:  PR[91,1] = PR[90,1] + -68.485;
   1:  PR[91,2] = PR[90,2] + 17.619;
   1:L PR[91] R[100]mm/sec CNT100;
   1:  PR[91,1] = PR[90,1] + -70.282;
   1:  PR[91,2] = PR[90,2] + 17.931;
   1:L PR[91] R[100]mm/sec CNT100;
   1:  PR[91,1] = PR[90,1] + -74.386;
   1:  PR[91,2] = PR[90,2] + 17.839;
   1:L PR[91] R[100]mm/sec CNT100;
   1:  PR[91,1] = PR[90,1] + -78.357;
   1:  PR[91,2] = PR[90,2] + 16.946;
   1:L PR[91] R[100]mm/sec CNT100;
   1:  PR[91,1] = PR[90,1] + -82.028;
   1:  PR[91,2] = PR[90,2] + 15.300;
   1:L PR[91] R[100]mm/sec CNT100;
   1:  PR[91,1] = PR[90,1] + -85.206;
   1:  PR[91,2] = PR[90,2] + 12.990;
   1:L PR[91] R[100]mm/sec CNT100;
   1:  PR[91,1] = PR[90,1] + -87.798;
   1:  PR[91,2] = PR[90,2] + 10.103;
   1:L PR[91] R[100]mm/sec CNT100;
   1:  PR[91,1] = PR[90,1] + -89.732;
   1:  PR[91,2] = PR[90,2] + 6.757;
   1:L PR[91] R[100]mm/sec CNT100;
   1:  PR[91,1] = PR[90,1] + -90.923;
   1:  PR[91,2] = PR[90,2] + 3.093;
   1:L PR[91] R[100]mm/sec CNT100;
   1:  PR[91,1] = PR[90,1] + -90.982;
   1:  PR[91,2] = PR[90,2] + 2.544;
   1:L PR[91] R[100]mm/sec CNT100;
   1:  PR[91,1] = PR[90,1] + -91.135;
   1:  PR[91,2] = PR[90,2] + 1.574;
   1:L PR[91] R[100]mm/sec CNT100;
   1:  PR[91,1] = PR[90,1] + -91.373;
   1:  PR[91,2] = PR[90,2] + -0.678;
   1:L PR[91] R[100]mm/sec CNT100;
   1:  PR[91,1] = PR[90,1] + -91.293;
   1:  PR[91,2] = PR[90,2] + -1.188;
   1:L PR[91] R[100]mm/sec CNT100;
   1:  PR[91,1] = PR[90,1] + -91.126;
   1:  PR[91,2] = PR[90,2] + -1.902;
   1:L PR[91] R[100]mm/sec CNT100;
   1:  PR[91,1] = PR[90,1] + -90.848;
   1:  PR[91,2] = PR[90,2] + -4.554;
   1:L PR[91] R[100]mm/sec CNT100;
   1:  PR[91,1] = PR[90,1] + -90.460;
   1:  PR[91,2] = PR[90,2] + -5.739;
   1:L PR[91] R[100]mm/sec CNT100;
   1:  PR[91,1] = PR[90,1] + -89.653;
   1:  PR[91,2] = PR[90,2] + -8.221;
   1:L PR[91] R[100]mm/sec CNT100;
   1:  PR[91,1] = PR[90,1] + -87.714;
   1:  PR[91,2] = PR[90,2] + -11.570;
   1:L PR[91] R[100]mm/sec CNT100;
   1:  PR[91,1] = PR[90,1] + -85.111;
   1:  PR[91,2] = PR[90,2] + -14.465;
   1:L PR[91] R[100]mm/sec CNT100;
   1:  PR[91,1] = PR[90,1] + -81.948;
   1:  PR[91,2] = PR[90,2] + -16.777;
   1:L PR[91] R[100]mm/sec CNT100;
   1:  PR[91,1] = PR[90,1] + -78.359;
   1:  PR[91,2] = PR[90,2] + -18.406;
   1:L PR[91] R[100]mm/sec CNT100;
   1:  PR[91,1] = PR[90,1] + -74.469;
   1:  PR[91,2] = PR[90,2] + -19.281;
   1:L PR[91] R[100]mm/sec CNT100;
   1:  PR[91,1] = PR[90,1] + -70.334;
   1:  PR[91,2] = PR[90,2] + -19.379;
   1:L PR[91] R[100]mm/sec CNT100;
   1:  PR[91,1] = PR[90,1] + -67.041;
   1:  PR[91,2] = PR[90,2] + -18.790;
   1:L PR[91] R[100]mm/sec CNT100;
   1:  PR[91,1] = PR[90,1] + -66.230;
   1:  PR[91,2] = PR[90,2] + -18.657;
   1:L PR[91] R[100]mm/sec CNT100;
   1:  PR[91,1] = PR[90,1] + -63.633;
   1:  PR[91,2] = PR[90,2] + -17.624;
   1:L PR[91] R[100]mm/sec CNT100;
   1:  PR[91,1] = PR[90,1] + -62.365;
   1:  PR[91,2] = PR[90,2] + -17.142;
   1:L PR[91] R[100]mm/sec CNT100;
   1:  PR[91,1] = PR[90,1] + -60.499;
   1:  PR[91,2] = PR[90,2] + -15.910;
   1:L PR[91] R[100]mm/sec CNT100;
   1:  PR[91,1] = PR[90,1] + -58.899;
   1:  PR[91,2] = PR[90,2] + -14.886;
   1:L PR[91] R[100]mm/sec CNT100;
   1:  PR[91,1] = PR[90,1] + -57.721;
   1:  PR[91,2] = PR[90,2] + -13.686;
   1:L PR[91] R[100]mm/sec CNT100;
   1:  PR[91,1] = PR[90,1] + -55.994;
   1:  PR[91,2] = PR[90,2] + -11.972;
   1:L PR[91] R[100]mm/sec CNT100;
   1:  PR[91,1] = PR[90,1] + -53.806;
   1:  PR[91,2] = PR[90,2] + -8.540;
   1:L PR[91] R[100]mm/sec CNT100;
   1:  PR[91,1] = PR[90,1] + -52.444;
   1:  PR[91,2] = PR[90,2] + -4.731;
   1:L PR[91] R[100]mm/sec CNT100TB   .50sec,CALL END_PUD;
   1:  PR[92] = PR[91];
   1:  PR[92,3] = PR[92,3] + 20;
   1:J PR[92] 10% FINE;
   1:  PR[91] = PR[90];
   1:  PR[91,1] = PR[90,1] + 65.665;
   1:  PR[91,2] = PR[90,2] + 18.026;
   1:  PR[91,3] = PR[90,3] + 30.095;
   1:  PR[92] = PR[91];
   1:  PR[92,3] = PR[92,3] + 20;
   1:J PR[92] 10% FINE;
   1:L PR[91] R[100]mm/sec CNT100;
   1:  CALL LASER_DRAHT_START;
   1:  PR[91,1] = PR[90,1] + 62.481;
   1:  PR[91,2] = PR[90,2] + 17.159;
   1:L PR[91] R[100]mm/sec CNT100;
   1:  PR[91,1] = PR[90,1] + 62.045;
   1:  PR[91,2] = PR[90,2] + 16.917;
   1:L PR[91] R[100]mm/sec CNT100;
   1:  PR[91,1] = PR[90,1] + 58.910;
   1:  PR[91,2] = PR[90,2] + 15.262;
   1:L PR[91] R[100]mm/sec CNT100;
   1:  PR[91,1] = PR[90,1] + 58.234;
   1:  PR[91,2] = PR[90,2] + 14.935;
   1:L PR[91] R[100]mm/sec CNT100;
   1:  PR[91,1] = PR[90,1] + 58.180;
   1:  PR[91,2] = PR[90,2] + 14.897;
   1:L PR[91] R[100]mm/sec CNT100;
   1:  PR[91,1] = PR[90,1] + 54.683;
   1:  PR[91,2] = PR[90,2] + 12.095;
   1:L PR[91] R[100]mm/sec CNT100;
   1:  PR[91,1] = PR[90,1] + 53.674;
   1:  PR[91,2] = PR[90,2] + 10.924;
   1:L PR[91] R[100]mm/sec CNT100;
   1:  PR[91,1] = PR[90,1] + 51.769;
   1:  PR[91,2] = PR[90,2] + 8.450;
   1:L PR[91] R[100]mm/sec CNT100;
   1:  PR[91,1] = PR[90,1] + 50.629;
   1:  PR[91,2] = PR[90,2] + 6.027;
   1:L PR[91] R[100]mm/sec CNT100;
   1:  PR[91,1] = PR[90,1] + 49.813;
   1:  PR[91,2] = PR[90,2] + 4.103;
   1:L PR[91] R[100]mm/sec CNT100;
   1:  PR[91,1] = PR[90,1] + 49.326;
   1:  PR[91,2] = PR[90,2] + 0.913;
   1:L PR[91] R[100]mm/sec CNT100;
   1:  PR[91,1] = PR[90,1] + 49.102;
   1:  PR[91,2] = PR[90,2] + -0.695;
   1:L PR[91] R[100]mm/sec CNT100;
   1:  PR[91,1] = PR[90,1] + 49.327;
   1:  PR[91,2] = PR[90,2] + -2.379;
   1:L PR[91] R[100]mm/sec CNT100;
   1:  PR[91,1] = PR[90,1] + 49.813;
   1:  PR[91,2] = PR[90,2] + -5.561;
   1:L PR[91] R[100]mm/sec CNT100;
   1:  PR[91,1] = PR[90,1] + 50.629;
   1:  PR[91,2] = PR[90,2] + -7.485;
   1:L PR[91] R[100]mm/sec CNT100;
   1:  PR[91,1] = PR[90,1] + 51.768;
   1:  PR[91,2] = PR[90,2] + -9.909;
   1:L PR[91] R[100]mm/sec CNT100;
   1:  PR[91,1] = PR[90,1] + 53.673;
   1:  PR[91,2] = PR[90,2] + -12.382;
   1:L PR[91] R[100]mm/sec CNT100;
   1:  PR[91,1] = PR[90,1] + 54.682;
   1:  PR[91,2] = PR[90,2] + -13.554;
   1:L PR[91] R[100]mm/sec CNT100;
   1:  PR[91,1] = PR[90,1] + 58.180;
   1:  PR[91,2] = PR[90,2] + -16.356;
   1:L PR[91] R[100]mm/sec CNT100;
   1:  PR[91,1] = PR[90,1] + 58.234;
   1:  PR[91,2] = PR[90,2] + -16.393;
   1:L PR[91] R[100]mm/sec CNT100;
   1:  PR[91,1] = PR[90,1] + 58.913;
   1:  PR[91,2] = PR[90,2] + -16.723;
   1:L PR[91] R[100]mm/sec CNT100;
   1:  PR[91,1] = PR[90,1] + 62.480;
   1:  PR[91,2] = PR[90,2] + -18.622;
   1:L PR[91] R[100]mm/sec CNT100;
   1:  PR[91,1] = PR[90,1] + 63.191;
   1:  PR[91,2] = PR[90,2] + -18.831;
   1:L PR[91] R[100]mm/sec CNT100;
   1:  PR[91,1] = PR[90,1] + 66.959;
   1:  PR[91,2] = PR[90,2] + -19.873;
   1:L PR[91] R[100]mm/sec CNT100;
   1:  PR[91,1] = PR[90,1] + 68.821;
   1:  PR[91,2] = PR[90,2] + -20.006;
   1:L PR[91] R[100]mm/sec CNT100;
   1:  PR[91,1] = PR[90,1] + 71.564;
   1:  PR[91,2] = PR[90,2] + -20.161;
   1:L PR[91] R[100]mm/sec CNT100;
   1:  PR[91,1] = PR[90,1] + 74.370;
   1:  PR[91,2] = PR[90,2] + -19.761;
   1:L PR[91] R[100]mm/sec CNT100;
   1:  PR[91,1] = PR[90,1] + 76.078;
   1:  PR[91,2] = PR[90,2] + -19.494;
   1:L PR[91] R[100]mm/sec CNT100;
   1:  PR[91,1] = PR[90,1] + 79.461;
   1:  PR[91,2] = PR[90,2] + -18.247;
   1:L PR[91] R[100]mm/sec CNT100;
   1:  PR[91,1] = PR[90,1] + 80.291;
   1:  PR[91,2] = PR[90,2] + -17.928;
   1:L PR[91] R[100]mm/sec CNT100;
   1:  PR[91,1] = PR[90,1] + 84.027;
   1:  PR[91,2] = PR[90,2] + -15.542;
   1:L PR[91] R[100]mm/sec CNT100;
   1:  PR[91,1] = PR[90,1] + 87.096;
   1:  PR[91,2] = PR[90,2] + -12.480;
   1:L PR[91] R[100]mm/sec CNT100;
   1:  PR[91,1] = PR[90,1] + 89.333;
   1:  PR[91,2] = PR[90,2] + -8.889;
   1:L PR[91] R[100]mm/sec CNT100;
   1:  PR[91,1] = PR[90,1] + 90.726;
   1:  PR[91,2] = PR[90,2] + -4.882;
   1:L PR[91] R[100]mm/sec CNT100;
   1:  PR[91,1] = PR[90,1] + 90.839;
   1:  PR[91,2] = PR[90,2] + -4.069;
   1:L PR[91] R[100]mm/sec CNT100;
   1:  PR[91,1] = PR[90,1] + 91.206;
   1:  PR[91,2] = PR[90,2] + -0.801;
   1:L PR[91] R[100]mm/sec CNT100;
   1:  PR[91,1] = PR[90,1] + 91.161;
   1:  PR[91,2] = PR[90,2] + -0.555;
   1:L PR[91] R[100]mm/sec CNT100;
   1:  PR[91,1] = PR[90,1] + 90.717;
   1:  PR[91,2] = PR[90,2] + 3.449;
   1:L PR[91] R[100]mm/sec CNT100;
   1:  PR[91,1] = PR[90,1] + 89.333;
   1:  PR[91,2] = PR[90,2] + 7.430;
   1:L PR[91] R[100]mm/sec CNT100;
   1:  PR[91,1] = PR[90,1] + 87.096;
   1:  PR[91,2] = PR[90,2] + 11.022;
   1:L PR[91] R[100]mm/sec CNT100;
   1:  PR[91,1] = PR[90,1] + 84.027;
   1:  PR[91,2] = PR[90,2] + 14.083;
   1:L PR[91] R[100]mm/sec CNT100;
   1:  PR[91,1] = PR[90,1] + 80.304;
   1:  PR[91,2] = PR[90,2] + 16.461;
   1:L PR[91] R[100]mm/sec CNT100;
   1:  PR[91,1] = PR[90,1] + 77.126;
   1:  PR[91,2] = PR[90,2] + 17.626;
   1:L PR[91] R[100]mm/sec CNT100;
   1:  PR[91,1] = PR[90,1] + 76.078;
   1:  PR[91,2] = PR[90,2] + 18.031;
   1:L PR[91] R[100]mm/sec CNT100;
   1:  PR[91,1] = PR[90,1] + 73.304;
   1:  PR[91,2] = PR[90,2] + 18.419;
   1:L PR[91] R[100]mm/sec CNT100;
   1:  PR[91,1] = PR[90,1] + 71.564;
   1:  PR[91,2] = PR[90,2] + 18.698;
   1:L PR[91] R[100]mm/sec CNT100;
   1:  PR[91,1] = PR[90,1] + 69.448;
   1:  PR[91,2] = PR[90,2] + 18.541;
   1:L PR[91] R[100]mm/sec CNT100;
   1:  PR[91,1] = PR[90,1] + 66.959;
   1:  PR[91,2] = PR[90,2] + 18.410;
   1:L PR[91] R[100]mm/sec CNT100;
   1:  PR[91,1] = PR[90,1] + 65.665;
   1:  PR[91,2] = PR[90,2] + 18.026;
   1:L PR[91] R[100]mm/sec CNT100TB   .50sec,CALL END_PUD;
   1:  PR[92] = PR[91];
   1:  PR[92,3] = PR[92,3] + 20;
   1:J PR[92] 10% FINE;
   1:  PR[91,1] = PR[90,1] + 42.274;
   1:  PR[91,2] = PR[90,2] + -7.577;
   1:  PR[92] = PR[91];
   1:  PR[92,3] = PR[92,3] + 20;
   1:J PR[92] 10% FINE;
   1:L PR[91] R[100]mm/sec CNT100;
   1:  CALL LASER_DRAHT_START;
   1:  PR[91,1] = PR[90,1] + 42.750;
   1:  PR[91,2] = PR[90,2] + -6.514;
   1:L PR[91] R[100]mm/sec CNT100;
   1:  PR[91,1] = PR[90,1] + 43.237;
   1:  PR[91,2] = PR[90,2] + -4.609;
   1:L PR[91] R[100]mm/sec CNT100;
   1:  PR[91,1] = PR[90,1] + 43.424;
   1:  PR[91,2] = PR[90,2] + -3.188;
   1:L PR[91] R[100]mm/sec CNT100;
   1:  PR[91,1] = PR[90,1] + 43.637;
   1:  PR[91,2] = PR[90,2] + -0.772;
   1:L PR[91] R[100]mm/sec CNT100;
   1:  PR[91,1] = PR[90,1] + 43.502;
   1:  PR[91,2] = PR[90,2] + 0.258;
   1:L PR[91] R[100]mm/sec CNT100;
   1:  PR[91,1] = PR[90,1] + 43.243;
   1:  PR[91,2] = PR[90,2] + 3.100;
   1:L PR[91] R[100]mm/sec CNT100;
   1:  PR[91,1] = PR[90,1] + 42.697;
   1:  PR[91,2] = PR[90,2] + 5.213;
   1:L PR[91] R[100]mm/sec CNT100;
   1:  PR[91,1] = PR[90,1] + 41.859;
   1:  PR[91,2] = PR[90,2] + 7.242;
   1:L PR[91] R[100]mm/sec CNT100;
   1:  PR[91,1] = PR[90,1] + 41.217;
   1:  PR[91,2] = PR[90,2] + 8.697;
   1:L PR[91] R[100]mm/sec CNT100;
   1:  PR[91,1] = PR[90,1] + 41.093;
   1:  PR[91,2] = PR[90,2] + 8.924;
   1:L PR[91] R[100]mm/sec CNT100;
   1:  PR[91,1] = PR[90,1] + 39.306;
   1:  PR[91,2] = PR[90,2] + 11.270;
   1:L PR[91] R[100]mm/sec CNT100;
   1:  PR[91,1] = PR[90,1] + 37.948;
   1:  PR[91,2] = PR[90,2] + 12.997;
   1:L PR[91] R[100]mm/sec CNT100;
   1:  PR[91,1] = PR[90,1] + 35.756;
   1:  PR[91,2] = PR[90,2] + 14.688;
   1:L PR[91] R[100]mm/sec CNT100;
   1:  PR[91,1] = PR[90,1] + 33.951;
   1:  PR[91,2] = PR[90,2] + 16.047;
   1:L PR[91] R[100]mm/sec CNT100;
   1:  PR[91,1] = PR[90,1] + 31.464;
   1:  PR[91,2] = PR[90,2] + 17.087;
   1:L PR[91] R[100]mm/sec CNT100;
   1:  PR[91,1] = PR[90,1] + 29.300;
   1:  PR[91,2] = PR[90,2] + 17.969;
   1:L PR[91] R[100]mm/sec CNT100;
   1:  PR[91,1] = PR[90,1] + 24.296;
   1:  PR[91,2] = PR[90,2] + 18.631;
   1:L PR[91] R[100]mm/sec CNT100;
   1:  PR[91,1] = PR[90,1] + 19.286;
   1:  PR[91,2] = PR[90,2] + 17.979;
   1:L PR[91] R[100]mm/sec CNT100;
   1:  PR[91,1] = PR[90,1] + 17.035;
   1:  PR[91,2] = PR[90,2] + 17.057;
   1:L PR[91] R[100]mm/sec CNT100;
   1:  PR[91,1] = PR[90,1] + 14.614;
   1:  PR[91,2] = PR[90,2] + 16.055;
   1:L PR[91] R[100]mm/sec CNT100;
   1:  PR[91,1] = PR[90,1] + 10.590;
   1:  PR[91,2] = PR[90,2] + 12.984;
   1:L PR[91] R[100]mm/sec CNT100;
   1:  PR[91,1] = PR[90,1] + 7.499;
   1:  PR[91,2] = PR[90,2] + 8.972;
   1:L PR[91] R[100]mm/sec CNT100;
   1:  PR[91,1] = PR[90,1] + 6.643;
   1:  PR[91,2] = PR[90,2] + 6.918;
   1:L PR[91] R[100]mm/sec CNT100;
   1:  PR[91,1] = PR[90,1] + 5.553;
   1:  PR[91,2] = PR[90,2] + 4.295;
   1:L PR[91] R[100]mm/sec CNT100;
   1:  PR[91,1] = PR[90,1] + 4.889;
   1:  PR[91,2] = PR[90,2] + -0.729;
   1:L PR[91] R[100]mm/sec CNT100;
   1:  PR[91,1] = PR[90,1] + 5.554;
   1:  PR[91,2] = PR[90,2] + -5.756;
   1:L PR[91] R[100]mm/sec CNT100;
   1:  PR[91,1] = PR[90,1] + 7.502;
   1:  PR[91,2] = PR[90,2] + -10.436;
   1:L PR[91] R[100]mm/sec CNT100;
   1:  PR[91,1] = PR[90,1] + 9.203;
   1:  PR[91,2] = PR[90,2] + -12.645;
   1:L PR[91] R[100]mm/sec CNT100;
   1:  PR[91,1] = PR[90,1] + 10.595;
   1:  PR[91,2] = PR[90,2] + -14.448;
   1:L PR[91] R[100]mm/sec CNT100;
   1:  PR[91,1] = PR[90,1] + 14.622;
   1:  PR[91,2] = PR[90,2] + -17.519;
   1:L PR[91] R[100]mm/sec CNT100;
   1:  PR[91,1] = PR[90,1] + 19.303;
   1:  PR[91,2] = PR[90,2] + -19.442;
   1:L PR[91] R[100]mm/sec CNT100;
   1:  PR[91,1] = PR[90,1] + 21.809;
   1:  PR[91,2] = PR[90,2] + -19.771;
   1:L PR[91] R[100]mm/sec CNT100;
   1:  PR[91,1] = PR[90,1] + 24.309;
   1:  PR[91,2] = PR[90,2] + -20.090;
   1:L PR[91] R[100]mm/sec CNT100;
   1:  PR[91,1] = PR[90,1] + 29.312;
   1:  PR[91,2] = PR[90,2] + -19.424;
   1:L PR[91] R[100]mm/sec CNT100;
   1:  PR[91,1] = PR[90,1] + 33.970;
   1:  PR[91,2] = PR[90,2] + -17.495;
   1:L PR[91] R[100]mm/sec CNT100;
   1:  PR[91,1] = PR[90,1] + 35.771;
   1:  PR[91,2] = PR[90,2] + -16.131;
   1:L PR[91] R[100]mm/sec CNT100;
   1:  PR[91,1] = PR[90,1] + 37.962;
   1:  PR[91,2] = PR[90,2] + -14.441;
   1:L PR[91] R[100]mm/sec CNT100;
   1:  PR[91,1] = PR[90,1] + 39.326;
   1:  PR[91,2] = PR[90,2] + -12.696;
   1:L PR[91] R[100]mm/sec CNT100;
   1:  PR[91,1] = PR[90,1] + 41.093;
   1:  PR[91,2] = PR[90,2] + -10.384;
   1:L PR[91] R[100]mm/sec CNT100;
   1:  PR[91,1] = PR[90,1] + 41.185;
   1:  PR[91,2] = PR[90,2] + -10.215;
   1:L PR[91] R[100]mm/sec CNT100;
   1:  PR[91,1] = PR[90,1] + 42.274;
   1:  PR[91,2] = PR[90,2] + -7.577;
   1:L PR[91] R[100]mm/sec CNT100TB   .50sec,CALL END_PUD;
   1:  PR[92] = PR[91];
   1:  PR[92,3] = PR[92,3] + 20;
   1:J PR[92] 10% FINE;
   1:  PR[91,1] = PR[90,1] + -5.269;
   1:  PR[91,2] = PR[90,2] + 7.364;
   1:  PR[92] = PR[91];
   1:  PR[92,3] = PR[92,3] + 20;
   1:J PR[92] 10% FINE;
   1:L PR[91] R[100]mm/sec CNT100;
   1:  CALL LASER_DRAHT_START;
   1:  PR[91,1] = PR[90,1] + -5.412;
   1:  PR[91,2] = PR[90,2] + 7.679;
   1:L PR[91] R[100]mm/sec CNT100;
   1:  PR[91,1] = PR[90,1] + -7.750;
   1:  PR[91,2] = PR[90,2] + 11.155;
   1:L PR[91] R[100]mm/sec CNT100;
   1:  PR[91,1] = PR[90,1] + -7.803;
   1:  PR[91,2] = PR[90,2] + 11.224;
   1:L PR[91] R[100]mm/sec CNT100;
   1:  PR[91,1] = PR[90,1] + -10.999;
   1:  PR[91,2] = PR[90,2] + 14.200;
   1:L PR[91] R[100]mm/sec CNT100;
   1:  PR[91,1] = PR[90,1] + -14.709;
   1:  PR[91,2] = PR[90,2] + 16.425;
   1:L PR[91] R[100]mm/sec CNT100;
   1:  PR[91,1] = PR[90,1] + -18.799;
   1:  PR[91,2] = PR[90,2] + 17.763;
   1:L PR[91] R[100]mm/sec CNT100;
   1:  PR[91,1] = PR[90,1] + -23.072;
   1:  PR[91,2] = PR[90,2] + 18.170;
   1:L PR[91] R[100]mm/sec CNT100;
   1:  PR[91,1] = PR[90,1] + -27.313;
   1:  PR[91,2] = PR[90,2] + 17.630;
   1:L PR[91] R[100]mm/sec CNT100;
   1:  PR[91,1] = PR[90,1] + -31.320;
   1:  PR[91,2] = PR[90,2] + 16.182;
   1:L PR[91] R[100]mm/sec CNT100;
   1:  PR[91,1] = PR[90,1] + -32.483;
   1:  PR[91,2] = PR[90,2] + 15.448;
   1:L PR[91] R[100]mm/sec CNT100;
   1:  PR[91,1] = PR[90,1] + -34.882;
   1:  PR[91,2] = PR[90,2] + 13.908;
   1:L PR[91] R[100]mm/sec CNT100;
   1:  PR[91,1] = PR[90,1] + -37.851;
   1:  PR[91,2] = PR[90,2] + 10.916;
   1:L PR[91] R[100]mm/sec CNT100;
   1:  PR[91,1] = PR[90,1] + -40.075;
   1:  PR[91,2] = PR[90,2] + 7.361;
   1:L PR[91] R[100]mm/sec CNT100;
   1:  PR[91,1] = PR[90,1] + -41.451;
   1:  PR[91,2] = PR[90,2] + 3.415;
   1:L PR[91] R[100]mm/sec CNT100;
   1:  PR[91,1] = PR[90,1] + -41.677;
   1:  PR[91,2] = PR[90,2] + 1.423;
   1:L PR[91] R[100]mm/sec CNT100;
   1:  PR[91,1] = PR[90,1] + -41.728;
   1:  PR[91,2] = PR[90,2] + 1.173;
   1:L PR[91] R[100]mm/sec CNT100;
   1:  PR[91,1] = PR[90,1] + -41.940;
   1:  PR[91,2] = PR[90,2] + -0.717;
   1:L PR[91] R[100]mm/sec CNT100;
   1:  PR[91,1] = PR[90,1] + -41.702;
   1:  PR[91,2] = PR[90,2] + -2.633;
   1:L PR[91] R[100]mm/sec CNT100;
   1:  PR[91,1] = PR[90,1] + -41.451;
   1:  PR[91,2] = PR[90,2] + -4.875;
   1:L PR[91] R[100]mm/sec CNT100;
   1:  PR[91,1] = PR[90,1] + -40.075;
   1:  PR[91,2] = PR[90,2] + -8.820;
   1:L PR[91] R[100]mm/sec CNT100;
   1:  PR[91,1] = PR[90,1] + -37.851;
   1:  PR[91,2] = PR[90,2] + -12.375;
   1:L PR[91] R[100]mm/sec CNT100;
   1:  PR[91,1] = PR[90,1] + -34.884;
   1:  PR[91,2] = PR[90,2] + -15.365;
   1:L PR[91] R[100]mm/sec CNT100;
   1:  PR[91,1] = PR[90,1] + -31.315;
   1:  PR[91,2] = PR[90,2] + -17.643;
   1:L PR[91] R[100]mm/sec CNT100;
   1:  PR[91,1] = PR[90,1] + -27.313;
   1:  PR[91,2] = PR[90,2] + -19.089;
   1:L PR[91] R[100]mm/sec CNT100;
   1:  PR[91,1] = PR[90,1] + -23.072;
   1:  PR[91,2] = PR[90,2] + -19.629;
   1:L PR[91] R[100]mm/sec CNT100;
   1:  PR[91,1] = PR[90,1] + -18.799;
   1:  PR[91,2] = PR[90,2] + -19.222;
   1:L PR[91] R[100]mm/sec CNT100;
   1:  PR[91,1] = PR[90,1] + -14.709;
   1:  PR[91,2] = PR[90,2] + -17.884;
   1:L PR[91] R[100]mm/sec CNT100;
   1:  PR[91,1] = PR[90,1] + -10.999;
   1:  PR[91,2] = PR[90,2] + -15.659;
   1:L PR[91] R[100]mm/sec CNT100;
   1:  PR[91,1] = PR[90,1] + -7.803;
   1:  PR[91,2] = PR[90,2] + -12.683;
   1:L PR[91] R[100]mm/sec CNT100;
   1:  PR[91,1] = PR[90,1] + -7.750;
   1:  PR[91,2] = PR[90,2] + -12.614;
   1:L PR[91] R[100]mm/sec CNT100;
   1:  PR[91,1] = PR[90,1] + -5.412;
   1:  PR[91,2] = PR[90,2] + -9.139;
   1:L PR[91] R[100]mm/sec CNT100;
   1:  PR[91,1] = PR[90,1] + -5.269;
   1:  PR[91,2] = PR[90,2] + -8.824;
   1:L PR[91] R[100]mm/sec CNT100;
   1:  PR[91,1] = PR[90,1] + -3.898;
   1:  PR[91,2] = PR[90,2] + -5.146;
   1:L PR[91] R[100]mm/sec CNT100;
   1:  PR[91,1] = PR[90,1] + -3.803;
   1:  PR[91,2] = PR[90,2] + -4.644;
   1:L PR[91] R[100]mm/sec CNT100;
   1:  PR[91,1] = PR[90,1] + -3.342;
   1:  PR[91,2] = PR[90,2] + -0.824;
   1:L PR[91] R[100]mm/sec CNT100;
   1:  PR[91,1] = PR[90,1] + -3.341;
   1:  PR[91,2] = PR[90,2] + -0.821;
   1:L PR[91] R[100]mm/sec CNT100;
   1:  PR[91,1] = PR[90,1] + -3.814;
   1:  PR[91,2] = PR[90,2] + 3.101;
   1:L PR[91] R[100]mm/sec CNT100;
   1:  PR[91,1] = PR[90,1] + -3.819;
   1:  PR[91,2] = PR[90,2] + 3.270;
   1:L PR[91] R[100]mm/sec CNT100;
   1:  PR[91,1] = PR[90,1] + -3.897;
   1:  PR[91,2] = PR[90,2] + 3.686;
   1:L PR[91] R[100]mm/sec CNT100;
   1:  PR[91,1] = PR[90,1] + -5.269;
   1:  PR[91,2] = PR[90,2] + 7.364;
   1:L PR[91] R[100]mm/sec CNT100TB   .50sec,CALL END_PUD;
   1:  PR[92] = PR[91];
   1:  PR[92,3] = PR[92,3] + 20;
   1:J PR[92] 10% FINE;
   1:  PR[91,1] = PR[90,1] + -65.835;
   1:  PR[91,2] = PR[90,2] + 17.309;
   1:  PR[92] = PR[91];
   1:  PR[92,3] = PR[92,3] + 20;
   1:J PR[92] 10% FINE;
   1:L PR[91] R[100]mm/sec CNT100;
   1:  CALL LASER_DRAHT_START;
   1:  PR[91,1] = PR[90,1] + -67.251;
   1:  PR[91,2] = PR[90,2] + 17.568;
   1:L PR[91] R[100]mm/sec CNT100;
   1:  PR[91,1] = PR[90,1] + -69.905;
   1:  PR[91,2] = PR[90,2] + 18.028;
   1:L PR[91] R[100]mm/sec CNT100;
   1:  PR[91,1] = PR[90,1] + -72.104;
   1:  PR[91,2] = PR[90,2] + 17.985;
   1:L PR[91] R[100]mm/sec CNT100;
   1:  PR[91,1] = PR[90,1] + -74.021;
   1:  PR[91,2] = PR[90,2] + 17.930;
   1:L PR[91] R[100]mm/sec CNT100;
   1:  PR[91,1] = PR[90,1] + -76.804;
   1:  PR[91,2] = PR[90,2] + 17.308;
   1:L PR[91] R[100]mm/sec CNT100;
   1:  PR[91,1] = PR[90,1] + -78.006;
   1:  PR[91,2] = PR[90,2] + 17.028;
   1:L PR[91] R[100]mm/sec CNT100;
   1:  PR[91,1] = PR[90,1] + -81.701;
   1:  PR[91,2] = PR[90,2] + 15.366;
   1:L PR[91] R[100]mm/sec CNT100;
   1:  PR[91,1] = PR[90,1] + -84.943;
   1:  PR[91,2] = PR[90,2] + 13.028;
   1:L PR[91] R[100]mm/sec CNT100;
   1:  PR[91,1] = PR[90,1] + -87.601;
   1:  PR[91,2] = PR[90,2] + 10.120;
   1:L PR[91] R[100]mm/sec CNT100;
   1:  PR[91,1] = PR[90,1] + -89.553;
   1:  PR[91,2] = PR[90,2] + 6.770;
   1:L PR[91] R[100]mm/sec CNT100;
   1:  PR[91,1] = PR[90,1] + -90.754;
   1:  PR[91,2] = PR[90,2] + 3.074;
   1:L PR[91] R[100]mm/sec CNT100;
   1:  PR[91,1] = PR[90,1] + -90.794;
   1:  PR[91,2] = PR[90,2] + 2.786;
   1:L PR[91] R[100]mm/sec CNT100;
   1:  PR[91,1] = PR[90,1] + -91.160;
   1:  PR[91,2] = PR[90,2] + -0.669;
   1:L PR[91] R[100]mm/sec CNT100;
   1:  PR[91,1] = PR[90,1] + -90.974;
   1:  PR[91,2] = PR[90,2] + -1.462;
   1:L PR[91] R[100]mm/sec CNT100;
   1:  PR[91,1] = PR[90,1] + -90.649;
   1:  PR[91,2] = PR[90,2] + -4.563;
   1:L PR[91] R[100]mm/sec CNT100;
   1:  PR[91,1] = PR[90,1] + -90.399;
   1:  PR[91,2] = PR[90,2] + -5.327;
   1:L PR[91] R[100]mm/sec CNT100;
   1:  PR[91,1] = PR[90,1] + -89.453;
   1:  PR[91,2] = PR[90,2] + -8.240;
   1:L PR[91] R[100]mm/sec CNT100;
   1:  PR[91,1] = PR[90,1] + -87.510;
   1:  PR[91,2] = PR[90,2] + -11.599;
   1:L PR[91] R[100]mm/sec CNT100;
   1:  PR[91,1] = PR[90,1] + -84.901;
   1:  PR[91,2] = PR[90,2] + -14.503;
   1:L PR[91] R[100]mm/sec CNT100;
   1:  PR[91,1] = PR[90,1] + -81.734;
   1:  PR[91,2] = PR[90,2] + -16.822;
   1:L PR[91] R[100]mm/sec CNT100;
   1:  PR[91,1] = PR[90,1] + -78.088;
   1:  PR[91,2] = PR[90,2] + -18.470;
   1:L PR[91] R[100]mm/sec CNT100;
   1:  PR[91,1] = PR[90,1] + -74.068;
   1:  PR[91,2] = PR[90,2] + -19.378;
   1:L PR[91] R[100]mm/sec CNT100;
   1:  PR[91,1] = PR[90,1] + -70.781;
   1:  PR[91,2] = PR[90,2] + -19.450;
   1:L PR[91] R[100]mm/sec CNT100;
   1:  PR[91,1] = PR[90,1] + -69.897;
   1:  PR[91,2] = PR[90,2] + -19.483;
   1:L PR[91] R[100]mm/sec CNT100;
   1:  PR[91,1] = PR[90,1] + -67.185;
   1:  PR[91,2] = PR[90,2] + -18.997;
   1:L PR[91] R[100]mm/sec CNT100;
   1:  PR[91,1] = PR[90,1] + -65.779;
   1:  PR[91,2] = PR[90,2] + -18.768;
   1:L PR[91] R[100]mm/sec CNT100;
   1:  PR[91,1] = PR[90,1] + -63.752;
   1:  PR[91,2] = PR[90,2] + -17.961;
   1:L PR[91] R[100]mm/sec CNT100;
   1:  PR[91,1] = PR[90,1] + -61.885;
   1:  PR[91,2] = PR[90,2] + -17.252;
   1:L PR[91] R[100]mm/sec CNT100;
   1:  PR[91,1] = PR[90,1] + -60.564;
   1:  PR[91,2] = PR[90,2] + -16.379;
   1:L PR[91] R[100]mm/sec CNT100;
   1:  PR[91,1] = PR[90,1] + -58.389;
   1:  PR[91,2] = PR[90,2] + -14.988;
   1:L PR[91] R[100]mm/sec CNT100;
   1:  PR[91,1] = PR[90,1] + -57.698;
   1:  PR[91,2] = PR[90,2] + -14.284;
   1:L PR[91] R[100]mm/sec CNT100;
   1:  PR[91,1] = PR[90,1] + -55.455;
   1:  PR[91,2] = PR[90,2] + -12.058;
   1:L PR[91] R[100]mm/sec CNT100;
   1:  PR[91,1] = PR[90,1] + -53.244;
   1:  PR[91,2] = PR[90,2] + -8.601;
   1:L PR[91] R[100]mm/sec CNT100;
   1:  PR[91,1] = PR[90,1] + -52.306;
   1:  PR[91,2] = PR[90,2] + -5.987;
   1:L PR[91] R[100]mm/sec CNT100;
   1:  PR[91,1] = PR[90,1] + -51.827;
   1:  PR[91,2] = PR[90,2] + -4.736;
   1:L PR[91] R[100]mm/sec CNT100;
   1:  PR[91,1] = PR[90,1] + -51.339;
   1:  PR[91,2] = PR[90,2] + -0.808;
   1:L PR[91] R[100]mm/sec CNT100;
   1:  PR[91,1] = PR[90,1] + -51.335;
   1:  PR[91,2] = PR[90,2] + -0.743;
   1:L PR[91] R[100]mm/sec CNT100;
   1:  PR[91,1] = PR[90,1] + -51.543;
   1:  PR[91,2] = PR[90,2] + 1.740;
   1:L PR[91] R[100]mm/sec CNT100;
   1:  PR[91,1] = PR[90,1] + -51.729;
   1:  PR[91,2] = PR[90,2] + 3.294;
   1:L PR[91] R[100]mm/sec CNT100;
   1:  PR[91,1] = PR[90,1] + -53.158;
   1:  PR[91,2] = PR[90,2] + 7.120;
   1:L PR[91] R[100]mm/sec CNT100;
   1:  PR[91,1] = PR[90,1] + -55.454;
   1:  PR[91,2] = PR[90,2] + 10.569;
   1:L PR[91] R[100]mm/sec CNT100;
   1:  PR[91,1] = PR[90,1] + -58.503;
   1:  PR[91,2] = PR[90,2] + 13.501;
   1:L PR[91] R[100]mm/sec CNT100;
   1:  PR[91,1] = PR[90,1] + -61.978;
   1:  PR[91,2] = PR[90,2] + 15.784;
   1:L PR[91] R[100]mm/sec CNT100;
   1:  PR[91,1] = PR[90,1] + -65.835;
   1:  PR[91,2] = PR[90,2] + 17.309;
   1:L PR[91] R[100]mm/sec CNT100TB   .50sec,CALL END_PUD;
   1:  PR[92] = PR[91];
   1:  PR[92,3] = PR[92,3] + 20;
   1:J PR[92] 10% FINE;
   1:  PR[91] = PR[90];
   1:  PR[91,1] = PR[90,1] + 54.067;
   1:  PR[91,2] = PR[90,2] + -13.931;
   1:  PR[91,3] = PR[90,3] + 31.395;
   1:  PR[92] = PR[91];
   1:  PR[92,3] = PR[92,3] + 20;
   1:J PR[92] 10% FINE;
   1:L PR[91] R[100]mm/sec CNT100;
   1:  CALL LASER_DRAHT_START;
   1:  PR[91,1] = PR[90,1] + 56.524;
   1:  PR[91,2] = PR[90,2] + -15.899;
   1:L PR[91] R[100]mm/sec CNT100;
   1:  PR[91,1] = PR[90,1] + 57.775;
   1:  PR[91,2] = PR[90,2] + -16.769;
   1:L PR[91] R[100]mm/sec CNT100;
   1:  PR[91,1] = PR[90,1] + 61.953;
   1:  PR[91,2] = PR[90,2] + -18.788;
   1:L PR[91] R[100]mm/sec CNT100;
   1:  PR[91,1] = PR[90,1] + 66.520;
   1:  PR[91,2] = PR[90,2] + -20.043;
   1:L PR[91] R[100]mm/sec CNT100;
   1:  PR[91,1] = PR[90,1] + 67.435;
   1:  PR[91,2] = PR[90,2] + -20.108;
   1:L PR[91] R[100]mm/sec CNT100;
   1:  PR[91,1] = PR[90,1] + 71.167;
   1:  PR[91,2] = PR[90,2] + -20.319;
   1:L PR[91] R[100]mm/sec CNT100;
   1:  PR[91,1] = PR[90,1] + 73.113;
   1:  PR[91,2] = PR[90,2] + -20.042;
   1:L PR[91] R[100]mm/sec CNT100;
   1:  PR[91,1] = PR[90,1] + 75.714;
   1:  PR[91,2] = PR[90,2] + -19.634;
   1:L PR[91] R[100]mm/sec CNT100;
   1:  PR[91,1] = PR[90,1] + 78.353;
   1:  PR[91,2] = PR[90,2] + -18.661;
   1:L PR[91] R[100]mm/sec CNT100;
   1:  PR[91,1] = PR[90,1] + 79.955;
   1:  PR[91,2] = PR[90,2] + -18.047;
   1:L PR[91] R[100]mm/sec CNT100;
   1:  PR[91,1] = PR[90,1] + 82.863;
   1:  PR[91,2] = PR[90,2] + -16.194;
   1:L PR[91] R[100]mm/sec CNT100;
   1:  PR[91,1] = PR[90,1] + 83.702;
   1:  PR[91,2] = PR[90,2] + -15.646;
   1:L PR[91] R[100]mm/sec CNT100;
   1:  PR[91,1] = PR[90,1] + 86.454;
   1:  PR[91,2] = PR[90,2] + -12.900;
   1:L PR[91] R[100]mm/sec CNT100;
   1:  PR[91,1] = PR[90,1] + 86.793;
   1:  PR[91,2] = PR[90,2] + -12.555;
   1:L PR[91] R[100]mm/sec CNT100;
   1:  PR[91,1] = PR[90,1] + 89.100;
   1:  PR[91,2] = PR[90,2] + -8.917;
   1:L PR[91] R[100]mm/sec CNT100;
   1:  PR[91,1] = PR[90,1] + 90.519;
   1:  PR[91,2] = PR[90,2] + -4.915;
   1:L PR[91] R[100]mm/sec CNT100;
   1:  PR[91,1] = PR[90,1] + 91.005;
   1:  PR[91,2] = PR[90,2] + -0.729;
   1:L PR[91] R[100]mm/sec CNT100;
   1:  PR[91,1] = PR[90,1] + 90.519;
   1:  PR[91,2] = PR[90,2] + 3.456;
   1:L PR[91] R[100]mm/sec CNT100;
   1:  PR[91,1] = PR[90,1] + 89.100;
   1:  PR[91,2] = PR[90,2] + 7.458;
   1:L PR[91] R[100]mm/sec CNT100;
   1:  PR[91,1] = PR[90,1] + 86.797;
   1:  PR[91,2] = PR[90,2] + 11.089;
   1:L PR[91] R[100]mm/sec CNT100;
   1:  PR[91,1] = PR[90,1] + 83.710;
   1:  PR[91,2] = PR[90,2] + 14.178;
   1:L PR[91] R[100]mm/sec CNT100;
   1:  PR[91,1] = PR[90,1] + 80.939;
   1:  PR[91,2] = PR[90,2] + 15.939;
   1:L PR[91] R[100]mm/sec CNT100;
   1:  PR[91,1] = PR[90,1] + 79.955;
   1:  PR[91,2] = PR[90,2] + 16.585;
   1:L PR[91] R[100]mm/sec CNT100;
   1:  PR[91,1] = PR[90,1] + 77.344;
   1:  PR[91,2] = PR[90,2] + 17.541;
   1:L PR[91] R[100]mm/sec CNT100;
   1:  PR[91,1] = PR[90,1] + 75.714;
   1:  PR[91,2] = PR[90,2] + 18.171;
   1:L PR[91] R[100]mm/sec CNT100;
   1:  PR[91,1] = PR[90,1] + 73.559;
   1:  PR[91,2] = PR[90,2] + 18.473;
   1:L PR[91] R[100]mm/sec CNT100;
   1:  PR[91,1] = PR[90,1] + 71.167;
   1:  PR[91,2] = PR[90,2] + 18.856;
   1:L PR[91] R[100]mm/sec CNT100;
   1:  PR[91,1] = PR[90,1] + 69.715;
   1:  PR[91,2] = PR[90,2] + 18.748;
   1:L PR[91] R[100]mm/sec CNT100;
   1:  PR[91,1] = PR[90,1] + 66.521;
   1:  PR[91,2] = PR[90,2] + 18.580;
   1:L PR[91] R[100]mm/sec CNT100;
   1:  PR[91,1] = PR[90,1] + 65.913;
   1:  PR[91,2] = PR[90,2] + 18.400;
   1:L PR[91] R[100]mm/sec CNT100;
   1:  PR[91,1] = PR[90,1] + 61.871;
   1:  PR[91,2] = PR[90,2] + 17.296;
   1:L PR[91] R[100]mm/sec CNT100;
   1:  PR[91,1] = PR[90,1] + 57.776;
   1:  PR[91,2] = PR[90,2] + 15.311;
   1:L PR[91] R[100]mm/sec CNT100;
   1:  PR[91,1] = PR[90,1] + 56.524;
   1:  PR[91,2] = PR[90,2] + 14.440;
   1:L PR[91] R[100]mm/sec CNT100;
   1:  PR[91,1] = PR[90,1] + 54.067;
   1:  PR[91,2] = PR[90,2] + 12.472;
   1:L PR[91] R[100]mm/sec CNT100;
   1:  PR[91,1] = PR[90,1] + 52.041;
   1:  PR[91,2] = PR[90,2] + 10.120;
   1:L PR[91] R[100]mm/sec CNT100;
   1:  PR[91,1] = PR[90,1] + 50.998;
   1:  PR[91,2] = PR[90,2] + 8.764;
   1:L PR[91] R[100]mm/sec CNT100;
   1:  PR[91,1] = PR[90,1] + 49.187;
   1:  PR[91,2] = PR[90,2] + 4.915;
   1:L PR[91] R[100]mm/sec CNT100;
   1:  PR[91,1] = PR[90,1] + 48.923;
   1:  PR[91,2] = PR[90,2] + 4.292;
   1:L PR[91] R[100]mm/sec CNT100;
   1:  PR[91,1] = PR[90,1] + 48.166;
   1:  PR[91,2] = PR[90,2] + -0.709;
   1:L PR[91] R[100]mm/sec CNT100;
   1:  PR[91,1] = PR[90,1] + 48.210;
   1:  PR[91,2] = PR[90,2] + -1.088;
   1:L PR[91] R[100]mm/sec CNT100;
   1:  PR[91,1] = PR[90,1] + 48.922;
   1:  PR[91,2] = PR[90,2] + -5.748;
   1:L PR[91] R[100]mm/sec CNT100;
   1:  PR[91,1] = PR[90,1] + 49.186;
   1:  PR[91,2] = PR[90,2] + -6.372;
   1:L PR[91] R[100]mm/sec CNT100;
   1:  PR[91,1] = PR[90,1] + 50.997;
   1:  PR[91,2] = PR[90,2] + -10.222;
   1:L PR[91] R[100]mm/sec CNT100;
   1:  PR[91,1] = PR[90,1] + 52.041;
   1:  PR[91,2] = PR[90,2] + -11.578;
   1:L PR[91] R[100]mm/sec CNT100;
   1:  PR[91,1] = PR[90,1] + 54.067;
   1:  PR[91,2] = PR[90,2] + -13.931;
   1:L PR[91] R[100]mm/sec CNT100TB   .50sec,CALL END_PUD;
   1:  PR[92] = PR[91];
   1:  PR[92,3] = PR[92,3] + 20;
   1:J PR[92] 10% FINE;
   1:  PR[91,1] = PR[90,1] + 41.310;
   1:  PR[91,2] = PR[90,2] + 8.698;
   1:  PR[92] = PR[91];
   1:  PR[92,3] = PR[92,3] + 20;
   1:J PR[92] 10% FINE;
   1:L PR[91] R[100]mm/sec CNT100;
   1:  CALL LASER_DRAHT_START;
   1:  PR[91,1] = PR[90,1] + 41.139;
   1:  PR[91,2] = PR[90,2] + 9.014;
   1:L PR[91] R[100]mm/sec CNT100;
   1:  PR[91,1] = PR[90,1] + 39.627;
   1:  PR[91,2] = PR[90,2] + 11.001;
   1:L PR[91] R[100]mm/sec CNT100;
   1:  PR[91,1] = PR[90,1] + 37.965;
   1:  PR[91,2] = PR[90,2] + 13.114;
   1:L PR[91] R[100]mm/sec CNT100;
   1:  PR[91,1] = PR[90,1] + 36.139;
   1:  PR[91,2] = PR[90,2] + 14.523;
   1:L PR[91] R[100]mm/sec CNT100;
   1:  PR[91,1] = PR[90,1] + 33.939;
   1:  PR[91,2] = PR[90,2] + 16.180;
   1:L PR[91] R[100]mm/sec CNT100;
   1:  PR[91,1] = PR[90,1] + 31.882;
   1:  PR[91,2] = PR[90,2] + 17.040;
   1:L PR[91] R[100]mm/sec CNT100;
   1:  PR[91,1] = PR[90,1] + 29.256;
   1:  PR[91,2] = PR[90,2] + 18.110;
   1:L PR[91] R[100]mm/sec CNT100;
   1:  PR[91,1] = PR[90,1] + 24.218;
   1:  PR[91,2] = PR[90,2] + 18.774;
   1:L PR[91] R[100]mm/sec CNT100;
   1:  PR[91,1] = PR[90,1] + 19.174;
   1:  PR[91,2] = PR[90,2] + 18.114;
   1:L PR[91] R[100]mm/sec CNT100;
   1:  PR[91,1] = PR[90,1] + 17.373;
   1:  PR[91,2] = PR[90,2] + 17.377;
   1:L PR[91] R[100]mm/sec CNT100;
   1:  PR[91,1] = PR[90,1] + 14.470;
   1:  PR[91,2] = PR[90,2] + 16.176;
   1:L PR[91] R[100]mm/sec CNT100;
   1:  PR[91,1] = PR[90,1] + 10.419;
   1:  PR[91,2] = PR[90,2] + 13.082;
   1:L PR[91] R[100]mm/sec CNT100;
   1:  PR[91,1] = PR[90,1] + 7.306;
   1:  PR[91,2] = PR[90,2] + 9.041;
   1:L PR[91] R[100]mm/sec CNT100;
   1:  PR[91,1] = PR[90,1] + 6.644;
   1:  PR[91,2] = PR[90,2] + 7.450;
   1:L PR[91] R[100]mm/sec CNT100;
   1:  PR[91,1] = PR[90,1] + 5.348;
   1:  PR[91,2] = PR[90,2] + 4.331;
   1:L PR[91] R[100]mm/sec CNT100;
   1:  PR[91,1] = PR[90,1] + 4.679;
   1:  PR[91,2] = PR[90,2] + -0.729;
   1:L PR[91] R[100]mm/sec CNT100;
   1:  PR[91,1] = PR[90,1] + 5.349;
   1:  PR[91,2] = PR[90,2] + -5.793;
   1:L PR[91] R[100]mm/sec CNT100;
   1:  PR[91,1] = PR[90,1] + 7.310;
   1:  PR[91,2] = PR[90,2] + -10.507;
   1:L PR[91] R[100]mm/sec CNT100;
   1:  PR[91,1] = PR[90,1] + 9.337;
   1:  PR[91,2] = PR[90,2] + -13.137;
   1:L PR[91] R[100]mm/sec CNT100;
   1:  PR[91,1] = PR[90,1] + 10.425;
   1:  PR[91,2] = PR[90,2] + -14.548;
   1:L PR[91] R[100]mm/sec CNT100;
   1:  PR[91,1] = PR[90,1] + 14.481;
   1:  PR[91,2] = PR[90,2] + -17.640;
   1:L PR[91] R[100]mm/sec CNT100;
   1:  PR[91,1] = PR[90,1] + 19.193;
   1:  PR[91,2] = PR[90,2] + -19.578;
   1:L PR[91] R[100]mm/sec CNT100;
   1:  PR[91,1] = PR[90,1] + 22.207;
   1:  PR[91,2] = PR[90,2] + -19.974;
   1:L PR[91] R[100]mm/sec CNT100;
   1:  PR[91,1] = PR[90,1] + 24.235;
   1:  PR[91,2] = PR[90,2] + -20.233;
   1:L PR[91] R[100]mm/sec CNT100;
   1:  PR[91,1] = PR[90,1] + 29.272;
   1:  PR[91,2] = PR[90,2] + -19.564;
   1:L PR[91] R[100]mm/sec CNT100;
   1:  PR[91,1] = PR[90,1] + 33.962;
   1:  PR[91,2] = PR[90,2] + -17.625;
   1:L PR[91] R[100]mm/sec CNT100;
   1:  PR[91,1] = PR[90,1] + 36.158;
   1:  PR[91,2] = PR[90,2] + -15.963;
   1:L PR[91] R[100]mm/sec CNT100;
   1:  PR[91,1] = PR[90,1] + 37.983;
   1:  PR[91,2] = PR[90,2] + -14.556;
   1:L PR[91] R[100]mm/sec CNT100;
   1:  PR[91,1] = PR[90,1] + 39.652;
   1:  PR[91,2] = PR[90,2] + -12.419;
   1:L PR[91] R[100]mm/sec CNT100;
   1:  PR[91,1] = PR[90,1] + 41.138;
   1:  PR[91,2] = PR[90,2] + -10.475;
   1:L PR[91] R[100]mm/sec CNT100;
   1:  PR[91,1] = PR[90,1] + 41.275;
   1:  PR[91,2] = PR[90,2] + -10.225;
   1:L PR[91] R[100]mm/sec CNT100;
   1:  PR[91,1] = PR[90,1] + 42.172;
   1:  PR[91,2] = PR[90,2] + -8.051;
   1:L PR[91] R[100]mm/sec CNT100;
   1:  PR[91,1] = PR[90,1] + 42.758;
   1:  PR[91,2] = PR[90,2] + -6.742;
   1:L PR[91] R[100]mm/sec CNT100;
   1:  PR[91,1] = PR[90,1] + 43.359;
   1:  PR[91,2] = PR[90,2] + -4.389;
   1:L PR[91] R[100]mm/sec CNT100;
   1:  PR[91,1] = PR[90,1] + 43.445;
   1:  PR[91,2] = PR[90,2] + -3.736;
   1:L PR[91] R[100]mm/sec CNT100;
   1:  PR[91,1] = PR[90,1] + 43.707;
   1:  PR[91,2] = PR[90,2] + -0.772;
   1:L PR[91] R[100]mm/sec CNT100;
   1:  PR[91,1] = PR[90,1] + 43.683;
   1:  PR[91,2] = PR[90,2] + -0.589;
   1:L PR[91] R[100]mm/sec CNT100;
   1:  PR[91,1] = PR[90,1] + 43.369;
   1:  PR[91,2] = PR[90,2] + 2.862;
   1:L PR[91] R[100]mm/sec CNT100;
   1:  PR[91,1] = PR[90,1] + 42.695;
   1:  PR[91,2] = PR[90,2] + 5.468;
   1:L PR[91] R[100]mm/sec CNT100;
   1:  PR[91,1] = PR[90,1] + 42.093;
   1:  PR[91,2] = PR[90,2] + 6.927;
   1:L PR[91] R[100]mm/sec CNT100;
   1:  PR[91,1] = PR[90,1] + 41.310;
   1:  PR[91,2] = PR[90,2] + 8.698;
   1:L PR[91] R[100]mm/sec CNT100TB   .50sec,CALL END_PUD;
   1:  PR[92] = PR[91];
   1:  PR[92,3] = PR[92,3] + 20;
   1:J PR[92] 10% FINE;
   1:  PR[91,1] = PR[90,1] + -6.984;
   1:  PR[91,2] = PR[90,2] + -12.298;
   1:  PR[92] = PR[91];
   1:  PR[92,3] = PR[92,3] + 20;
   1:J PR[92] 10% FINE;
   1:L PR[91] R[100]mm/sec CNT100;
   1:  CALL LASER_DRAHT_START;
   1:  PR[91,1] = PR[90,1] + -5.016;
   1:  PR[91,2] = PR[90,2] + -9.371;
   1:L PR[91] R[100]mm/sec CNT100;
   1:  PR[91,1] = PR[90,1] + -4.586;
   1:  PR[91,2] = PR[90,2] + -8.422;
   1:L PR[91] R[100]mm/sec CNT100;
   1:  PR[91,1] = PR[90,1] + -3.447;
   1:  PR[91,2] = PR[90,2] + -5.368;
   1:L PR[91] R[100]mm/sec CNT100;
   1:  PR[91,1] = PR[90,1] + -3.223;
   1:  PR[91,2] = PR[90,2] + -4.180;
   1:L PR[91] R[100]mm/sec CNT100;
   1:  PR[91,1] = PR[90,1] + -2.843;
   1:  PR[91,2] = PR[90,2] + -1.030;
   1:L PR[91] R[100]mm/sec CNT100;
   1:  PR[91,1] = PR[90,1] + -2.837;
   1:  PR[91,2] = PR[90,2] + -0.821;
   1:L PR[91] R[100]mm/sec CNT100;
   1:  PR[91,1] = PR[90,1] + -3.226;
   1:  PR[91,2] = PR[90,2] + 2.415;
   1:L PR[91] R[100]mm/sec CNT100;
   1:  PR[91,1] = PR[90,1] + -3.239;
   1:  PR[91,2] = PR[90,2] + 2.803;
   1:L PR[91] R[100]mm/sec CNT100;
   1:  PR[91,1] = PR[90,1] + -3.445;
   1:  PR[91,2] = PR[90,2] + 3.905;
   1:L PR[91] R[100]mm/sec CNT100;
   1:  PR[91,1] = PR[90,1] + -4.585;
   1:  PR[91,2] = PR[90,2] + 6.960;
   1:L PR[91] R[100]mm/sec CNT100;
   1:  PR[91,1] = PR[90,1] + -5.014;
   1:  PR[91,2] = PR[90,2] + 7.909;
   1:L PR[91] R[100]mm/sec CNT100;
   1:  PR[91,1] = PR[90,1] + -6.983;
   1:  PR[91,2] = PR[90,2] + 10.836;
   1:L PR[91] R[100]mm/sec CNT100;
   1:  PR[91,1] = PR[90,1] + -7.457;
   1:  PR[91,2] = PR[90,2] + 11.450;
   1:L PR[91] R[100]mm/sec CNT100;
   1:  PR[91,1] = PR[90,1] + -10.305;
   1:  PR[91,2] = PR[90,2] + 14.095;
   1:L PR[91] R[100]mm/sec CNT100;
   1:  PR[91,1] = PR[90,1] + -10.633;
   1:  PR[91,2] = PR[90,2] + 14.361;
   1:L PR[91] R[100]mm/sec CNT100;
   1:  PR[91,1] = PR[90,1] + -14.364;
   1:  PR[91,2] = PR[90,2] + 16.511;
   1:L PR[91] R[100]mm/sec CNT100;
   1:  PR[91,1] = PR[90,1] + -14.377;
   1:  PR[91,2] = PR[90,2] + 16.517;
   1:L PR[91] R[100]mm/sec CNT100;
   1:  PR[91,1] = PR[90,1] + -16.694;
   1:  PR[91,2] = PR[90,2] + 17.235;
   1:L PR[91] R[100]mm/sec CNT100;
   1:  PR[91,1] = PR[90,1] + -18.585;
   1:  PR[91,2] = PR[90,2] + 17.853;
   1:L PR[91] R[100]mm/sec CNT100;
   1:  PR[91,1] = PR[90,1] + -22.887;
   1:  PR[91,2] = PR[90,2] + 18.257;
   1:L PR[91] R[100]mm/sec CNT100;
   1:  PR[91,1] = PR[90,1] + -23.181;
   1:  PR[91,2] = PR[90,2] + 18.222;
   1:L PR[91] R[100]mm/sec CNT100;
   1:  PR[91,1] = PR[90,1] + -27.137;
   1:  PR[91,2] = PR[90,2] + 17.710;
   1:L PR[91] R[100]mm/sec CNT100;
   1:  PR[91,1] = PR[90,1] + -31.156;
   1:  PR[91,2] = PR[90,2] + 16.254;
   1:L PR[91] R[100]mm/sec CNT100;
   1:  PR[91,1] = PR[90,1] + -34.738;
   1:  PR[91,2] = PR[90,2] + 13.964;
   1:L PR[91] R[100]mm/sec CNT100;
   1:  PR[91,1] = PR[90,1] + -37.714;
   1:  PR[91,2] = PR[90,2] + 10.961;
   1:L PR[91] R[100]mm/sec CNT100;
   1:  PR[91,1] = PR[90,1] + -39.945;
   1:  PR[91,2] = PR[90,2] + 7.391;
   1:L PR[91] R[100]mm/sec CNT100;
   1:  PR[91,1] = PR[90,1] + -41.325;
   1:  PR[91,2] = PR[90,2] + 3.430;
   1:L PR[91] R[100]mm/sec CNT100;
   1:  PR[91,1] = PR[90,1] + -41.504;
   1:  PR[91,2] = PR[90,2] + 1.857;
   1:L PR[91] R[100]mm/sec CNT100;
   1:  PR[91,1] = PR[90,1] + -41.545;
   1:  PR[91,2] = PR[90,2] + 1.656;
   1:L PR[91] R[100]mm/sec CNT100;
   1:  PR[91,1] = PR[90,1] + -41.811;
   1:  PR[91,2] = PR[90,2] + -0.717;
   1:L PR[91] R[100]mm/sec CNT100;
   1:  PR[91,1] = PR[90,1] + -41.624;
   1:  PR[91,2] = PR[90,2] + -2.220;
   1:L PR[91] R[100]mm/sec CNT100;
   1:  PR[91,1] = PR[90,1] + -41.325;
   1:  PR[91,2] = PR[90,2] + -4.890;
   1:L PR[91] R[100]mm/sec CNT100;
   1:  PR[91,1] = PR[90,1] + -39.945;
   1:  PR[91,2] = PR[90,2] + -8.850;
   1:L PR[91] R[100]mm/sec CNT100;
   1:  PR[91,1] = PR[90,1] + -37.714;
   1:  PR[91,2] = PR[90,2] + -12.419;
   1:L PR[91] R[100]mm/sec CNT100;
   1:  PR[91,1] = PR[90,1] + -34.738;
   1:  PR[91,2] = PR[90,2] + -15.423;
   1:L PR[91] R[100]mm/sec CNT100;
   1:  PR[91,1] = PR[90,1] + -31.156;
   1:  PR[91,2] = PR[90,2] + -17.713;
   1:L PR[91] R[100]mm/sec CNT100;
   1:  PR[91,1] = PR[90,1] + -27.138;
   1:  PR[91,2] = PR[90,2] + -19.169;
   1:L PR[91] R[100]mm/sec CNT100;
   1:  PR[91,1] = PR[90,1] + -22.878;
   1:  PR[91,2] = PR[90,2] + -19.715;
   1:L PR[91] R[100]mm/sec CNT100;
   1:  PR[91,1] = PR[90,1] + -18.585;
   1:  PR[91,2] = PR[90,2] + -19.311;
   1:L PR[91] R[100]mm/sec CNT100;
   1:  PR[91,1] = PR[90,1] + -16.694;
   1:  PR[91,2] = PR[90,2] + -18.694;
   1:L PR[91] R[100]mm/sec CNT100;
   1:  PR[91,1] = PR[90,1] + -14.376;
   1:  PR[91,2] = PR[90,2] + -17.976;
   1:L PR[91] R[100]mm/sec CNT100;
   1:  PR[91,1] = PR[90,1] + -14.364;
   1:  PR[91,2] = PR[90,2] + -17.970;
   1:L PR[91] R[100]mm/sec CNT100;
   1:  PR[91,1] = PR[90,1] + -10.634;
   1:  PR[91,2] = PR[90,2] + -15.821;
   1:L PR[91] R[100]mm/sec CNT100;
   1:  PR[91,1] = PR[90,1] + -10.307;
   1:  PR[91,2] = PR[90,2] + -15.555;
   1:L PR[91] R[100]mm/sec CNT100;
   1:  PR[91,1] = PR[90,1] + -7.459;
   1:  PR[91,2] = PR[90,2] + -12.910;
   1:L PR[91] R[100]mm/sec CNT100;
   1:  PR[91,1] = PR[90,1] + -6.984;
   1:  PR[91,2] = PR[90,2] + -12.298;
   1:L PR[91] R[100]mm/sec CNT100TB   .50sec,CALL END_PUD;
   1:  PR[92] = PR[91];
   1:  PR[92,3] = PR[92,3] + 20;
   1:J PR[92] 10% FINE;
   1:  PR[91,1] = PR[90,1] + -50.624;
   1:  PR[91,2] = PR[90,2] + -1.776;
   1:  PR[92] = PR[91];
   1:  PR[92,3] = PR[92,3] + 20;
   1:J PR[92] 10% FINE;
   1:L PR[91] R[100]mm/sec CNT100;
   1:  CALL LASER_DRAHT_START;
   1:  PR[91,1] = PR[90,1] + -50.552;
   1:  PR[91,2] = PR[90,2] + -0.743;
   1:L PR[91] R[100]mm/sec CNT100;
   1:  PR[91,1] = PR[90,1] + -50.671;
   1:  PR[91,2] = PR[90,2] + 0.667;
   1:L PR[91] R[100]mm/sec CNT100;
   1:  PR[91,1] = PR[90,1] + -50.990;
   1:  PR[91,2] = PR[90,2] + 3.333;
   1:L PR[91] R[100]mm/sec CNT100;
   1:  PR[91,1] = PR[90,1] + -52.439;
   1:  PR[91,2] = PR[90,2] + 7.197;
   1:L PR[91] R[100]mm/sec CNT100;
   1:  PR[91,1] = PR[90,1] + -53.729;
   1:  PR[91,2] = PR[90,2] + 9.141;
   1:L PR[91] R[100]mm/sec CNT100;
   1:  PR[91,1] = PR[90,1] + -54.759;
   1:  PR[91,2] = PR[90,2] + 10.668;
   1:L PR[91] R[100]mm/sec CNT100;
   1:  PR[91,1] = PR[90,1] + -57.832;
   1:  PR[91,2] = PR[90,2] + 13.604;
   1:L PR[91] R[100]mm/sec CNT100;
   1:  PR[91,1] = PR[90,1] + -61.506;
   1:  PR[91,2] = PR[90,2] + 15.875;
   1:L PR[91] R[100]mm/sec CNT100;
   1:  PR[91,1] = PR[90,1] + -65.421;
   1:  PR[91,2] = PR[90,2] + 17.406;
   1:L PR[91] R[100]mm/sec CNT100;
   1:  PR[91,1] = PR[90,1] + -69.521;
   1:  PR[91,2] = PR[90,2] + 18.124;
   1:L PR[91] R[100]mm/sec CNT100;
   1:  PR[91,1] = PR[90,1] + -73.660;
   1:  PR[91,2] = PR[90,2] + 18.018;
   1:L PR[91] R[100]mm/sec CNT100;
   1:  PR[91,1] = PR[90,1] + -77.665;
   1:  PR[91,2] = PR[90,2] + 17.105;
   1:L PR[91] R[100]mm/sec CNT100;
   1:  PR[91,1] = PR[90,1] + -81.369;
   1:  PR[91,2] = PR[90,2] + 15.433;
   1:L PR[91] R[100]mm/sec CNT100;
   1:  PR[91,1] = PR[90,1] + -84.621;
   1:  PR[91,2] = PR[90,2] + 13.083;
   1:L PR[91] R[100]mm/sec CNT100;
   1:  PR[91,1] = PR[90,1] + -87.291;
   1:  PR[91,2] = PR[90,2] + 10.158;
   1:L PR[91] R[100]mm/sec CNT100;
   1:  PR[91,1] = PR[90,1] + -89.275;
   1:  PR[91,2] = PR[90,2] + 6.786;
   1:L PR[91] R[100]mm/sec CNT100;
   1:  PR[91,1] = PR[90,1] + -90.495;
   1:  PR[91,2] = PR[90,2] + 3.105;
   1:L PR[91] R[100]mm/sec CNT100;
   1:  PR[91,1] = PR[90,1] + -90.905;
   1:  PR[91,2] = PR[90,2] + -0.673;
   1:L PR[91] R[100]mm/sec CNT100;
   1:  PR[91,1] = PR[90,1] + -90.823;
   1:  PR[91,2] = PR[90,2] + -1.023;
   1:L PR[91] R[100]mm/sec CNT100;
   1:  PR[91,1] = PR[90,1] + -90.451;
   1:  PR[91,2] = PR[90,2] + -4.573;
   1:L PR[91] R[100]mm/sec CNT100;
   1:  PR[91,1] = PR[90,1] + -90.339;
   1:  PR[91,2] = PR[90,2] + -4.915;
   1:L PR[91] R[100]mm/sec CNT100;
   1:  PR[91,1] = PR[90,1] + -89.252;
   1:  PR[91,2] = PR[90,2] + -8.259;
   1:L PR[91] R[100]mm/sec CNT100;
   1:  PR[91,1] = PR[90,1] + -87.305;
   1:  PR[91,2] = PR[90,2] + -11.628;
   1:L PR[91] R[100]mm/sec CNT100;
   1:  PR[91,1] = PR[90,1] + -84.698;
   1:  PR[91,2] = PR[90,2] + -14.534;
   1:L PR[91] R[100]mm/sec CNT100;
   1:  PR[91,1] = PR[90,1] + -81.441;
   1:  PR[91,2] = PR[90,2] + -16.878;
   1:L PR[91] R[100]mm/sec CNT100;
   1:  PR[91,1] = PR[90,1] + -77.708;
   1:  PR[91,2] = PR[90,2] + -18.554;
   1:L PR[91] R[100]mm/sec CNT100;
   1:  PR[91,1] = PR[90,1] + -74.560;
   1:  PR[91,2] = PR[90,2] + -19.259;
   1:L PR[91] R[100]mm/sec CNT100;
   1:  PR[91,1] = PR[90,1] + -73.654;
   1:  PR[91,2] = PR[90,2] + -19.475;
   1:L PR[91] R[100]mm/sec CNT100;
   1:  PR[91,1] = PR[90,1] + -70.925;
   1:  PR[91,2] = PR[90,2] + -19.535;
   1:L PR[91] R[100]mm/sec CNT100;
   1:  PR[91,1] = PR[90,1] + -69.472;
   1:  PR[91,2] = PR[90,2] + -19.588;
   1:L PR[91] R[100]mm/sec CNT100;
   1:  PR[91,1] = PR[90,1] + -67.329;
   1:  PR[91,2] = PR[90,2] + -19.205;
   1:L PR[91] R[100]mm/sec CNT100;
   1:  PR[91,1] = PR[90,1] + -65.328;
   1:  PR[91,2] = PR[90,2] + -18.879;
   1:L PR[91] R[100]mm/sec CNT100;
   1:  PR[91,1] = PR[90,1] + -63.871;
   1:  PR[91,2] = PR[90,2] + -18.299;
   1:L PR[91] R[100]mm/sec CNT100;
   1:  PR[91,1] = PR[90,1] + -61.406;
   1:  PR[91,2] = PR[90,2] + -17.361;
   1:L PR[91] R[100]mm/sec CNT100;
   1:  PR[91,1] = PR[90,1] + -60.629;
   1:  PR[91,2] = PR[90,2] + -16.848;
   1:L PR[91] R[100]mm/sec CNT100;
   1:  PR[91,1] = PR[90,1] + -57.871;
   1:  PR[91,2] = PR[90,2] + -15.084;
   1:L PR[91] R[100]mm/sec CNT100;
   1:  PR[91,1] = PR[90,1] + -55.179;
   1:  PR[91,2] = PR[90,2] + -12.403;
   1:L PR[91] R[100]mm/sec CNT100;
   1:  PR[91,1] = PR[90,1] + -54.850;
   1:  PR[91,2] = PR[90,2] + -12.098;
   1:L PR[91] R[100]mm/sec CNT100;
   1:  PR[91,1] = PR[90,1] + -52.476;
   1:  PR[91,2] = PR[90,2] + -8.631;
   1:L PR[91] R[100]mm/sec CNT100;
   1:  PR[91,1] = PR[90,1] + -50.998;
   1:  PR[91,2] = PR[90,2] + -4.779;
   1:L PR[91] R[100]mm/sec CNT100;
   1:  PR[91,1] = PR[90,1] + -50.624;
